IF bAlarmInit THEN
    bAlarmInit := FALSE; 
	fbSourceInfo.Clear();
	fbSourceInfo.sName:=wsLiteral_TO_UTF8(wsStationName);//'Machine';
	fbSourceInfo.nId:=iStationIndex;//83
	// Alarm_0610	610	Error	Siłownik przeciągania | Blokada wysunięcia - sprawdź czujnik lub odblokuj  
    arfbAlarm[0].CreateEx(stEventEntry := TC_EVENTS.AlarmClass.Alarm_0610, bWithConfirmation:= FALSE,  ipSourceInfo:= fbSourceInfo); 
	// Alarm_0611	611	Error	Siłownik przeciągania | Blokada wsunięcia - sprawdź czujnik lub odblokuj  
	arfbAlarm[1].CreateEx(stEventEntry := TC_EVENTS.AlarmClass.Alarm_0611, bWithConfirmation:= FALSE,  ipSourceInfo:= fbSourceInfo);
	// Alarm_0612	612	Error	Banda końcowa | Blokada wysunięcia - sprawdź czujnik lub odblokuj  
	arfbAlarm[2].CreateEx(stEventEntry := TC_EVENTS.AlarmClass.Alarm_0612, bWithConfirmation:= FALSE,  ipSourceInfo:= fbSourceInfo);
	// Alarm_0613	613	Error	Szlaban | Blokada wysunięcia - sprawdź czujnik lub odblokuj  
	arfbAlarm[3].CreateEx(stEventEntry := TC_EVENTS.AlarmClass.Alarm_0613, bWithConfirmation:= FALSE,  ipSourceInfo:= fbSourceInfo);
	// Alarm_0614	614	Error	Bład czujników przed przeciąganiem - sprawdź ułożenie formatek
	arfbAlarm[4].CreateEx(stEventEntry := TC_EVENTS.AlarmClass.Alarm_0614, bWithConfirmation:= FALSE,  ipSourceInfo:= fbSourceInfo);
	// Alarm_0615	615	Error	Bład czujników za przeciąganiem - sprawdź ułożenie formatek
	arfbAlarm[5].CreateEx(stEventEntry := TC_EVENTS.AlarmClass.Alarm_0615, bWithConfirmation:= FALSE,  ipSourceInfo:= fbSourceInfo);
	
END_IF

//CZYTANIE STATUSÓW
bStateError										:= (eState=E_Station.eError) OR (eState=E_Station.eResetting) OR NOT bEstop OR bIgnoreError;
tonEstopDelay									(IN:=bEStop,	PT:=T#4S);

IF bEnable AND tonEstopDelay.Q THEN
	// Alarm_0610	610	Error	Siłownik przeciągania | Blokada wysunięcia - sprawdź czujnik lub odblokuj  
	tonbDragOnSensor	(IN:= bDragActuator AND NOT bDragOnSensor	, PT:=T#2S);
	IF tonbDragOnSensor.Q THEN
		bHomingDone									:= FALSE;	
		//arfbAlarm[0].ipArguments.Clear() .AddString(stDrag.stError.sNcError);
		IF NOT arfbAlarm[0].bActive THEN
			arfbAlarm[0].Raise(nTimeStamp:=0);
		END_IF
	ELSE	
		IF  arfbAlarm[0].bActive AND bReset THEN
			arfbAlarm[0].Clear(nTimeStamp:=0, bResetConfirmation:= FALSE);
		END_IF	
	END_IF
	// Alarm_0611	611	Error	Siłownik przeciągania | Blokada wsunięcia - sprawdź czujnik lub odblokuj  
	tonbDragOffSensor	(IN:= NOT bDragActuator AND NOT bDragOffSensor	, PT:=T#2S);
	IF tonbDragOffSensor.Q THEN
		IF NOT arfbAlarm[1].bActive THEN
			arfbAlarm[1].Raise(nTimeStamp:=0);
		END_IF
	ELSE	
		IF  arfbAlarm[1].bActive AND bReset THEN
			arfbAlarm[1].Clear(nTimeStamp:=0, bResetConfirmation:= FALSE);
		END_IF	
	END_IF	
	// Alarm_0612	612	Error	Banda końcowa | Blokada wysunięcia - sprawdź czujnik lub odblokuj  
	tonbStoperOnSensor	(IN:= bStoperActuator AND NOT bStoperOnSensor	, PT:=T#2S);
	IF tonbStoperOnSensor.Q THEN
		IF NOT arfbAlarm[2].bActive THEN
			arfbAlarm[2].Raise(nTimeStamp:=0);
		END_IF
	ELSE	
		IF  arfbAlarm[2].bActive AND bReset THEN
			arfbAlarm[2].Clear(nTimeStamp:=0, bResetConfirmation:= FALSE);
		END_IF	
	END_IF	
	// Alarm_0613	613	Error	Szlaban | Blokada wysunięcia - sprawdź czujnik lub odblokuj  
	tonbGateSensor	(IN:= bGateActuator AND NOT bGateOnSensor	, PT:=T#2S);
	IF tonbGateSensor.Q THEN
		IF NOT arfbAlarm[3].bActive THEN
			arfbAlarm[3].Raise(nTimeStamp:=0);
		END_IF
	ELSE	
		IF  arfbAlarm[3].bActive AND bReset THEN
			arfbAlarm[3].Clear(nTimeStamp:=0, bResetConfirmation:= FALSE);
		END_IF	
	END_IF	
	// Alarm_0614	614	Error	Bład czujników przed przeciąganiem - sprawdź ułożenie formatek
	tonBeforeSensor	(IN:= NOT bFirstFormSensor AND bSecondFormSensor AND bConveyorBeforeRunning, PT:=T#20S);
	IF tonBeforeSensor.Q THEN
		IF NOT arfbAlarm[4].bActive THEN
			arfbAlarm[4].Raise(nTimeStamp:=0);
		END_IF
	ELSE	
		IF  arfbAlarm[4].bActive AND bReset THEN
			arfbAlarm[4].Clear(nTimeStamp:=0, bResetConfirmation:= FALSE);
		END_IF	
	END_IF	
	// Alarm_0615	615	Error	Bład czujników za przeciąganiem - sprawdź ułożenie formatek
	tonAfterSensor	(IN:= bAfterSensor AND bConveyorAfterRunning, PT:=T#20S);
	IF tonAfterSensor.Q THEN
		IF NOT arfbAlarm[5].bActive THEN
			arfbAlarm[5].Raise(nTimeStamp:=0);
		END_IF
	ELSE	
		IF  arfbAlarm[5].bActive AND bReset THEN
			arfbAlarm[5].Clear(nTimeStamp:=0, bResetConfirmation:= FALSE);
		END_IF	
	END_IF	
ELSE
	bError := FALSE;
END_IF

//******************PRZEJŚCIE DO eERROR*****************************

IF bError AND  NOT bStateError THEN
	eState 									:= E_Station.eError;
END_IF

//****************WYŚWIETLANIE STATUSU BLEDU************************
(*Wyświetlanie błedu na wyjściu*)
bError							:= FALSE;
FOR nAlarmNumerator := 0 TO 19 DO
	bError						:= bError OR arfbAlarm[nAlarmNumerator].bActive;
END_FOR

(*Przepisywanie nazwy stacji*)
sErrorStationName 							:= WSTRING_TO_STRING(wsStationName);
END_ACTION

ACTION Homing:


IF bHoming THEN // Bazowanie - podjazd do góry i ustawienie obrotu
	CASE iHomingCase OF
	
	0: 
		bHomingDone								:= FALSE;                                       		
		bDragActuator							:= FALSE;	
		bStoperActuator							:= TRUE; 	
		bGateActuator							:= FALSE;
			
		iHomingCase								:= 10;
	
	10: 
		iHomingCase								:= 20;
		
	20: 
		iHomingCase								:= 30;
		
		
	30:
		iHomingCase								:= 40;
		
	40:
		iHomingCase								:= 50;
	
	50: 
		iHomingCase								:= 60;
		
	60: 
		iHomingCase								:= 70;
	
	70:                             	
		iHomingCase								:= 80;

	80:
		iHomingCase								:= 100;

	100: //Zbazowano	
		iHomingCase								:= 0;
		eState									:= E_Station.eHomingDone;
	
	END_CASE
END_IF	
IF bHeightSet THEN

	bDragActuator								:= FALSE;	
	bStoperActuator								:= TRUE;
	bGateActuator								:= FALSE;
	eState										:= E_Station.eHomingDone;
		
END_IF
END_ACTION

ACTION Limits:
(*Wywowyłanie na początku*)


(*Prędkość zakręcania*)


(*Inny parametr*)
//...
END_ACTION

ACTION ManualMovements:

IF NOT bRun AND NOT bPrepare AND bManualMovement THEN
	bDragActuator							:=	bManualDragActuator;			
	bStoperActuator							:=	bManualStoperActuator;	
	bGateActuator							:=	bManualGateActuator;	
ELSE
	bManualDragActuator						:=	FALSE;		
	bManualStoperActuator					:=	TRUE;	
	bManualGateActuator						:=	FALSE;		
END_IF
	
IF bHoming OR bHeightSet THEN
	eState									:=	E_Station.eHoming;	
END_IF                                                	
                                                      	
Running();

IF NOT bRun AND NOT bPrepare THEN
	bCycleDone 								:= FALSE;
	bCycleNotDone 							:= FALSE;	
END_IF
END_ACTION

ACTION ResetAll:
(*****Reset bloczka*****)
IF bEnable THEN
	IF eState <> E_Station.eDisabled AND eState <> E_Station.ePreparingToDisable THEN
		IF bResetCycle THEN
			bResetCycleOn						:= TRUE;
			eState								:= E_Station.ePreparingToReady;
		END_IF
	END_IF
END_IF


IF bResetCycleOn THEN
	
	ResetCommands();
	eRunningState							:= E_DragStationState.eReady;	
	eState 				 					:= E_Station.eReady;

END_IF
END_ACTION

ACTION ResetCommands:
//KAsowanie komend ruchu 
                                                          	
bManualDragActuator								:=	FALSE;		
bManualStoperActuator							:=	FALSE;	
bManualGateActuator								:=	FALSE;	
                                                        	
bDragActuator									:=	FALSE;	
bStoperActuator									:=	TRUE;	
bGateActuator									:=	FALSE;
                                                          	
bResetCycleOn									:=	FALSE;	

iHomingCase										:=	0;
//bCycleDone								   	:=	FALSE;
END_ACTION

ACTION Running:
	
CASE eRunningState OF
	
	E_DragStationState.eDisabled:
		eRunningState								:= E_DragStationState.eReady; 
	
	E_DragStationState.eReady:

			//bDragActuator						:=	FALSE;
			//bStoperActuator					:=	TRUE;
			//bGateActuator						:=	FALSE;
			IF (bRun OR bPrepare) AND NOT bCycleDone THEN   
				eRunningState					:=	E_DragStationState.ePreparingToMove; 
       		END_IF

// Sygnal przygotowania do przeciaganiecia formatek		
	E_DragStationState.ePreparingToMove:
		bGateActuator							:=	TRUE;
		IF bGateOnSensor THEN
			eRunningState						:=	E_DragStationState.eLifting;
		END_IF
		
// Podnoszenie widel do przeciągania i sprawdzenie czy trafiły w otwór		
	E_DragStationState.eLifting:
	
		bStoperActuator							:=	FALSE;		
		IF NOT bStoperOnSensor AND bRun AND tonRunningLifting.Q THEN
			eRunningState						:=	E_DragStationState.eDraging;	
		END_IF
//  
	E_DragStationState.ePrepareToDrag:
		;
	
// Przeciąganie formatek
	E_DragStationState.eDraging:
	
		bDragActuator						:=	TRUE;
		IF bDragOnSensor THEN //100MS
			eRunningState							:= E_DragStationState.eDragingDone;
		END_IF

	E_DragStationState.eDragingDone:

		eRunningState							:= E_DragStationState.eEndingOfDrag;
	
	E_DragStationState.eEndingOfDrag:
		bDragActuator								:=	FALSE;
		IF bDragOffSensor THEN
			bStoperActuator							:=	TRUE;
			bGateActuator							:=	FALSE;				
			eRunningState							:= E_DragStationState.eEndingOfDragDone;
		END_IF	
		
	E_DragStationState.eEndingOfDragDone:
		
		eRunningState								:= E_DragStationState.eLowering;
	
	E_DragStationState.eLowering:
	
		eRunningState							:= E_DragStationState.eDraged;
	
	E_DragStationState.eDraged:
			
		eRunningState							:= E_DragStationState.eDragedDone;
		
	E_DragStationState.eDragedDone:
	
		bCycleDone									:= TRUE;	
		eRunningState								:= E_DragStationState.eReady;	
		
END_CASE
END_ACTION

ACTION Signals:

tonPreparingToReady		(IN:=	eState = E_Station.ePreparingToReady			,PT:= T#3S);
tonResetting			(IN:=	eState = E_Station.eResetting					,PT:= T#200MS);
tonHoming				(IN:=	eState = E_Station.eHoming						,PT:= T#1S);
rtResetCommands			(CLK:=	eState = E_Station.eReady 						,Q=>); 

tonRunningDraging		(IN:=	eRunningState = E_DragStationState.eDraging		,PT:= T#100MS);	//bylo 100
tonRunningLifting		(IN:=	eRunningState = E_DragStationState.eLifting		,PT:= T#100MS);	//bylo 100

tonRunningeEndingOfDrag	(IN:=	eRunningState = E_DragStationState.eEndingOfDrag 
								,PT:= T#5MS);								//100ms t#200ms

//Opóżnienie wysuwania przeciągania
tonNotDragActuatorDelay	(IN:=	NOT bDragActuator					,PT:=T#150MS);
END_ACTION

ACTION Statistics:
rtrigCycleTimerRead(CLK:=bCycleDone);
IF rtrigCycleTimerRead.Q THEN
	tCycleTime:=tonCycleTimer.ET;
END_IF
tonCycleTimer(IN:= eRunningState>E_DragStationState.eReady, PT:=T#1D);
END_ACTION

END_FUNCTION_BLOCK

// ---- POUs/P17_TurnTables.TcPOU
(*
Nazwa:			P14_TurnTable
Opis:			Stacja stołu obrotowego
Wersja:			v0.2
Data:			2024-11-06
Autor:			DP
Urzadzenia:		
Konfiguracja:	
Info:
- 4 wersja z safety po EC

*)
PROGRAM P17_TurnTables
VAR_INPUT
	IbExitTurnTableAfterSensor 			:BOOL;
	IbExitTurnTablePackageSensor 	AT %I*	:BOOL;		
END_VAR
VAR
	
	(*********STOL ODBIERAJACY*******************)
	
	tonIbExitTurnTable1Working		: TON;
	fbTurnTable						: FB_MitsubishiInverter; 	//Bloczek do obsługi falownika stołu obrotewego
	eTurnTableState					: E_Station;
	eTurnTableRunningState			: E_ConveyorState;
	fbTurnTableState				: FB_State;

	uiTurnTableSW					AT %I*: UINT;
	uiTurnTableActualVelocity		AT %I*: UDINT;
	uiTurnTableCW  					AT %Q*: UINT;
	udiTurnTableVelocity			AT %Q*: UDINT;	
	
	tonIbTurnTableCycleStopButton	: TON;
	bExitTurnTableCmdStartDelay		: BOOL;
	tonbExitTurnTableCmdStartDelay	: TON;
	
	//fbExitConveyor					: FB_LenzeInverter;
	fbExitConveyor					: FB_MitsubishiInverter;
	QnExitConveyorVelocitySV 		AT %Q*: UDINT; 		
	InExitConveyorVelocityCV 		AT %I*: UDINT;	
	InExitConveyorSTW 				AT %I*: UINT; 
	QnExitConveyorConvCTW 			AT %Q*: UINT;  			
	InExitConveyorErrorCode 		AT %I*:UINT;			

	fbExitTurnTableGate				: FB_Gate;				// Bloczek obsługi gata	
	QbExitTurnTableGate 			: BOOL; 				// Wyjście sterujące szlabanem stołu odbiorczego
	
	
	tonbExitTurnTableCmdStart		: TON;
	tonIbExitTurnTableAfterSensor	: TON;
	tonbExitTurnTableGateRunOn		: TON;
	tonbExitTurnTableGateRunOff		: TON;	
	
	fbExitConveyorGate				: FB_Gate;				
	QbExitConveyorGate 				AT %Q*: BOOL;			
	IbExitConveyorGateAfterSensor 	AT %I*: BOOL;		//Blizej szlabanu
	IbExitConveyorGateAfterSensor2 	AT %I*: BOOL;		//Dalej szlabanu
	
	
END_VAR

aTurnTable();
aConveyor();
aConveyorGate();
aTurnTableGate();
aTurnTableGateLogic();
(*
tonIbTurnTableCycleStopButton	(IN:=NOT IbTurnTableCycleStopButton AND bExitTurnTableCmdStart AND NOT (P00_PackML.fbPMLAuto.ePMLState = Tc3_PackML.E_PMLState.ePMLState_EXECUTE), PT:=T#10MS);
IF tonIbTurnTableCycleStopButton.Q THEN
	bExitTurnTableCmdStartDelay	:=	TRUE;
END_IF
IF bExitTurnTableCmdStartDelay THEN
	bExitTurnTableCmdStart	:=	FALSE;
END_IF
tonbExitTurnTableCmdStartDelay		(IN:= bExitTurnTableCmdStartDelay, PT:=T#5S);
IF 	tonbExitTurnTableCmdStartDelay.Q THEN
	bExitTurnTableCmdStartDelay	:=	FALSE;
END_IF
*)

IbTurnTableMotorOK							;
IbTurnTableEmergencyStopButtonPressed	;
IbTurnTableCycleStartButton				;
IbTurnTableCycleStopButton				;
										;

P00_Signalization.QbTurnTableStartLamp;							
P00_Signalization.QbTurnTableResetLamp;

ACTION aConveyor:
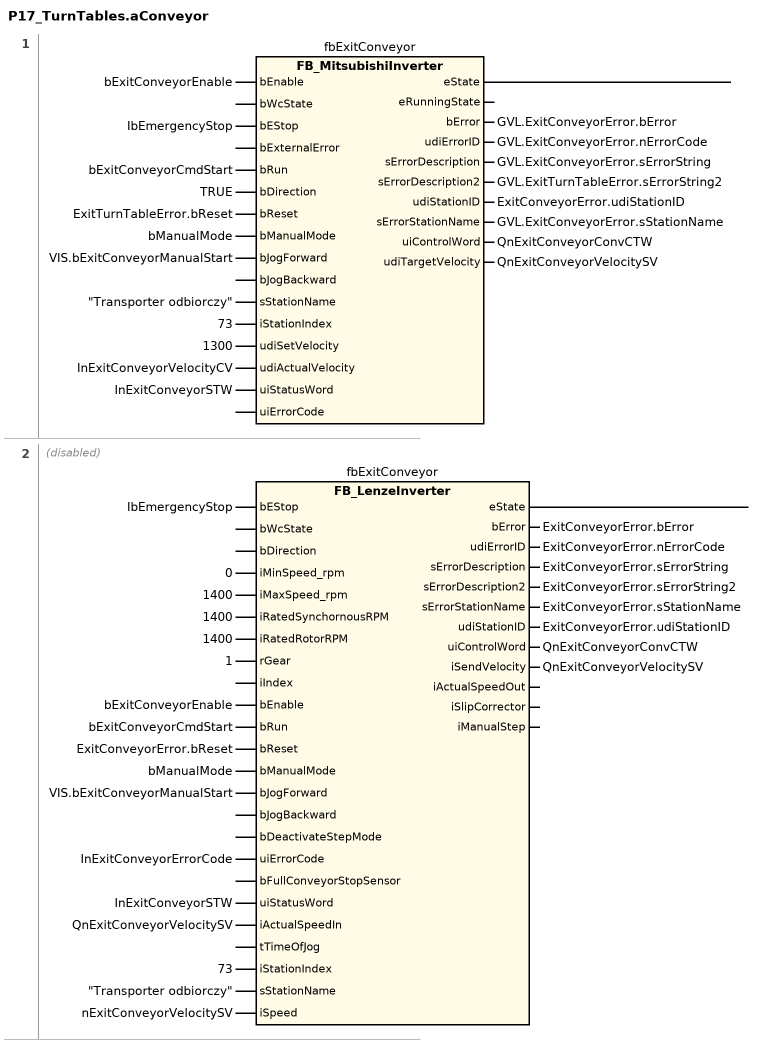
// NETWORK 1
fbExitConveyor(
    bEnable := bExitConveyorEnable,
    bEStop := IbEmergencyStop,
    bRun := bExitConveyorCmdStart,
    bDirection := TRUE,
    bReset := ExitTurnTableError.bReset,
    bManualMode := bManualMode,
    bJogForward := VIS.bExitConveyorManualStart,
    sStationName := "Transporter odbiorczy",
    iStationIndex := 73,
    udiSetVelocity := 1300,
    udiActualVelocity := InExitConveyorVelocityCV,
    uiStatusWord := InExitConveyorSTW,
    bError => GVL.ExitConveyorError.bError,
    udiErrorID => GVL.ExitConveyorError.nErrorCode,
    sErrorDescription => GVL.ExitConveyorError.sErrorString,
    sErrorDescription2 => GVL.ExitTurnTableError.sErrorString2,
    udiStationID => ExitConveyorError.udiStationID,
    sErrorStationName => GVL.ExitConveyorError.sStationName,
    uiControlWord => QnExitConveyorConvCTW,
    udiTargetVelocity => QnExitConveyorVelocitySV); // FB_MitsubishiInverter

// NETWORK 2 (disabled)
// fbExitConveyor(
//     bEStop := IbEmergencyStop,
//     iMinSpeed_rpm := 0,
//     iMaxSpeed_rpm := 1400,
//     iRatedSynchornousRPM := 1400,
//     iRatedRotorRPM := 1400,
//     rGear := 1,
//     bEnable := bExitConveyorEnable,
//     bRun := bExitConveyorCmdStart,
//     bReset := ExitConveyorError.bReset,
//     bManualMode := bManualMode,
//     bJogForward := VIS.bExitConveyorManualStart,
//     uiErrorCode := InExitConveyorErrorCode,
//     uiStatusWord := InExitConveyorSTW,
//     iActualSpeedIn := QnExitConveyorVelocitySV,
//     iStationIndex := 73,
//     sStationName := "Transporter odbiorczy",
//     iSpeed := nExitConveyorVelocitySV,
//     bError => ExitConveyorError.bError,
//     udiErrorID => ExitConveyorError.nErrorCode,
//     sErrorDescription => ExitConveyorError.sErrorString,
//     sErrorDescription2 => ExitConveyorError.sErrorString2,
//     sErrorStationName => ExitConveyorError.sStationName,
//     udiStationID => ExitConveyorError.udiStationID,
//     uiControlWord => QnExitConveyorConvCTW,
//     iSendVelocity => QnExitConveyorVelocitySV); // FB_LenzeInverter
END_ACTION

ACTION aConveyorGate:
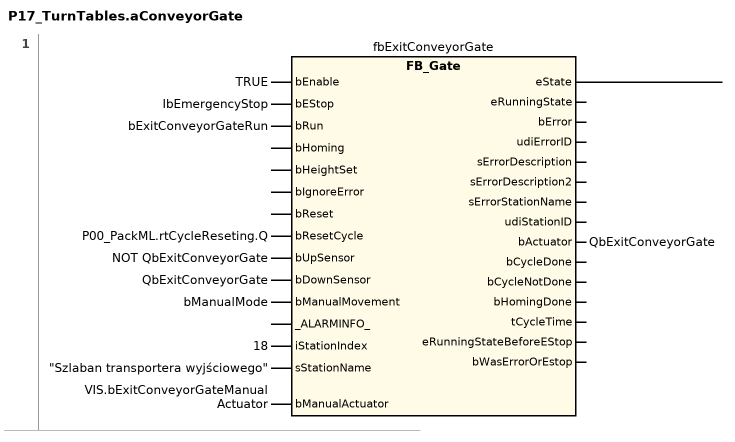
// NETWORK 1
fbExitConveyorGate(
    bEnable := TRUE,
    bEStop := IbEmergencyStop,
    bRun := bExitConveyorGateRun,
    bResetCycle := P00_PackML.rtCycleReseting.Q,
    bUpSensor := NOT QbExitConveyorGate,
    bDownSensor := QbExitConveyorGate,
    bManualMovement := bManualMode,
    iStationIndex := 18,
    sStationName := "Szlaban transportera wyjściowego",
    bManualActuator := VIS.bExitConveyorGateManualActuator,
    bActuator => QbExitConveyorGate); // FB_Gate
END_ACTION

ACTION aTurntable:
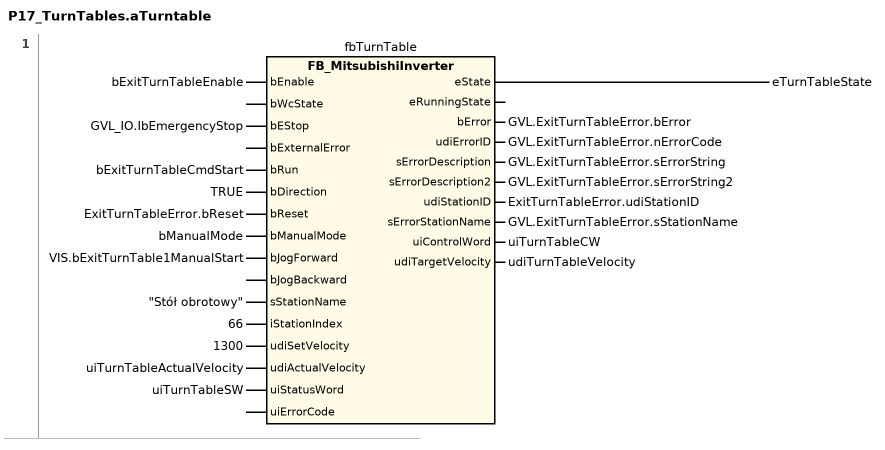
// NETWORK 1
fbTurnTable(
    bEnable := bExitTurnTableEnable,
    bEStop := GVL_IO.IbEmergencyStop,
    bRun := bExitTurnTableCmdStart,
    bDirection := TRUE,
    bReset := ExitTurnTableError.bReset,
    bManualMode := bManualMode,
    bJogForward := VIS.bExitTurnTable1ManualStart,
    sStationName := "Stół obrotowy",
    iStationIndex := 66,
    udiSetVelocity := 1300,
    udiActualVelocity := uiTurnTableActualVelocity,
    uiStatusWord := uiTurnTableSW,
    bError => GVL.ExitTurnTableError.bError,
    udiErrorID => GVL.ExitTurnTableError.nErrorCode,
    sErrorDescription => GVL.ExitTurnTableError.sErrorString,
    sErrorDescription2 => GVL.ExitTurnTableError.sErrorString2,
    udiStationID => ExitTurnTableError.udiStationID,
    sErrorStationName => GVL.ExitTurnTableError.sStationName,
    uiControlWord => uiTurnTableCW,
    udiTargetVelocity => udiTurnTableVelocity); // FB_MitsubishiInverter
eTurnTableState := fbTurnTable.eState;
END_ACTION

ACTION aTurntableGate:
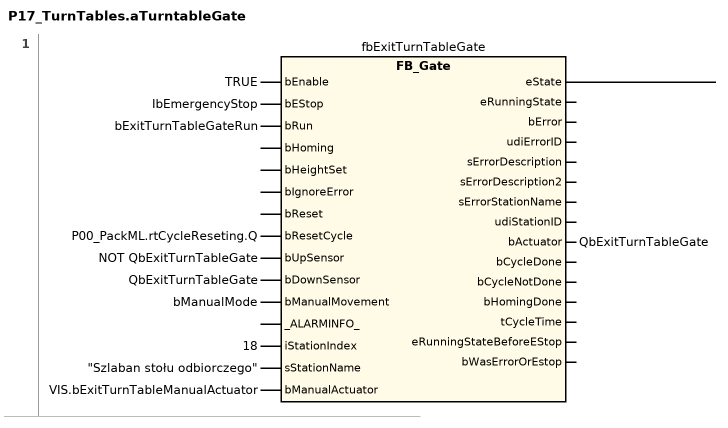
// NETWORK 1
fbExitTurnTableGate(
    bEnable := TRUE,
    bEStop := IbEmergencyStop,
    bRun := bExitTurnTableGateRun,
    bResetCycle := P00_PackML.rtCycleReseting.Q,
    bUpSensor := NOT QbExitTurnTableGate,
    bDownSensor := QbExitTurnTableGate,
    bManualMovement := bManualMode,
    iStationIndex := 18,
    sStationName := "Szlaban stołu odbiorczego",
    bManualActuator := VIS.bExitTurnTableManualActuator,
    bActuator => QbExitTurnTableGate); // FB_Gate
END_ACTION

ACTION aTurnTableGateLogic:
//Jeżeli stół pracuje 
bExitTurnTableCmdStart;
//To ruszaj szlabanem
bExitTurnTableGateRun;
//Czujnik na szlabanie etykieciarki:
IbExitTurnTableAfterSensor;

tonbExitTurnTableCmdStart		(IN:=bExitTurnTableCmdStart,											PT:=T#3S);
tonIbExitTurnTableAfterSensor	(IN:=IbExitTurnTableAfterSensor,										PT:=T#3S);
tonbExitTurnTableGateRunOn		(IN:=bExitTurnTableGateRun ,											PT:=T#5S);
tonbExitTurnTableGateRunOff		(IN:=NOT bExitTurnTableGateRun AND tonIbExitTurnTableAfterSensor.Q,		PT:=T#5S);//bylo 1

IF tonbExitTurnTableCmdStart.Q THEN
	bExitTurnTableGateRun R= tonbExitTurnTableGateRunOn.Q;
	bExitTurnTableGateRun S= tonbExitTurnTableGateRunOff.Q;	
END_IF
END_ACTION

END_PROGRAM

// ---- POUs/FB/FB_LenzeInverter.TcPOU
////////////////////////////////////////////////////////////////////////////////////////////////////////////
(*	TKMatik
	Blok funkcyjny, sterujacy falownikiem firmy Lenze model:i550
	v.1.3 16.01.2019
	v.1.4 22.08.2019
	v.1.5 29.07.2020
	Wymagane pliki: E_Station (ENUM)
	Data modyfikacji: 29.07.2020
	
	--->Obsluga bloku:
	Blok umozliwia sterownie falownikiem Lenze i550 w trybie manulanym i automatycznym
	*TRYB AUTOMATYCZNY*
	Po podaniu sygnalu wysokiego na wejscie bEnable rozoczyna sie procedura uruchamiania falownika
	Wejscie bRun umozliwiaja odpowiednio uruchomienie silnika i jego zatrzymanie 
	Wejscie bReset umozliwa wykonanie procedury resetu bloku i bledu falownika
	Wejscia iMinSpeed_rpm oraz iMaxSpeed_rpm pozwalaja na programowe ograniczenie obrotow silnika
	Wejscie iSpeed sluzy zadawania wartosci predkosci
	Mozliwa jest rowniez zmiana kierunku obrotow silnika przy pomocy wejscia bDirection
	*TRYB MANULANY*
	Sterowanie w trybie manulanym opiera sie o wykrywanie czasu przyciniecia przyciku
	Dla krotkiego przycisniecia wykonywany jest ruch silnika o krok ktorego czas musi byc zadany na wejscie bloku - opcje ta mozna dezaktywowac wejsciem bStepModeNotActive
	Dla dlugiego przycisniecia ruch jest wykonywany do czasu zaprzestania naciskania przycisku
	
	
	Wejscia bloku, ktore nalezy polinkowac ze zmiennymi falownika:
		-uiErrorCode
		-uiStatusWord
		-ActualSpeed 
	Wyjscia bloku, ktore nalezy polinkowac ze zmiennymi falownika:
		-uiControlWord
		-iSendVelocity
*)
////////////////////////////////////////////////////////////////////////////////////////////////////////////

FUNCTION_BLOCK FB_LenzeInverter

VAR_INPUT
	bEStop														: BOOL;													// Pozwolenie na prace bloku z SAFETY (TRUE-maszyna gotowa do pracy FALSE-brak pozolenia na prace)
	bWcState													: BOOL;													// Zmienna WcState - TRUE w przypadku odebrania niewlasciwej ramki EtherCAT
	bDirection													: BOOL;													// Kierunek obrotow silnika 
	iMinSpeed_rpm												: INT				:= 1000;							// Minimalna prędkość obrotowa
	iMaxSpeed_rpm												: INT				:= 2840;							// Maksymalna prędkość obrotowa
	iRatedSynchornousRPM										: INT				:= 3000;							// Predkosc synchorniczna (wzor: RatedSynchronousRPM = 60 * Frequency / NumberOfPolePair)
	iRatedRotorRPM												: INT				:= 2840;							// Znamionowe obroty silnika
	rGear														: REAL;													// Przekładnia
	iIndex														: INT;													// Indeks falownika
	bEnable														: BOOL;													// Uruchomienie bloku
	bRun														: BOOL;													// Komenda na uruchomienie 
	bReset														: BOOL;													// Reset falownika po bledzie
	bManualMode													: BOOL;													// Tryb manualny
	bJogForward													: BOOL;													// Komenda na ruch w kierunku dodatnim 
	bJogBackward												: BOOL;													// Komenda na ruch w kierunku ujemnym 
	bDeactivateStepMode											: BOOL;													// Zmienna dezaktywujaca przesuwanie silnika o krok po nacisnieciu JOGa
	uiErrorCode 				(*Devices*)						: UINT;													// Kod bledu falownika
	bFullConveyorStopSensor										: BOOL;													// Zatrzymanie transportera ze względu zapełnienia
	uiStatusWord				(*Devices*)						: UINT;													// Status wysylany z falownika
	iActualSpeedIn				(*Devices*)						: INT;													// Zmienna z falownika przepisana na wyjscie do zmiennej QiActualSpeed
	tTimeOfJog													: TIME				:= T#2S;
	iStationIndex												: UDINT;												// Numer stacji 
	sStationName												: WSTRING;												// Nazwa stacji
	iSpeed														: INT;													// Predkosc zadana przypisana do zmiennej Qn_SV wysylanej do falownika  
END_VAR                                                                         			                    		
VAR_OUTPUT                                                                      			                    		
	eState														: E_Station;											// Stan pracy bloku
	
	bError														: BOOL;													// Blad falownika
	udiErrorID													: UDINT;												// Nr błędu bloku funkcyjnego
	sErrorDescription											: STRING(200);											// Opis błędu
	sErrorDescription2											: STRING(200);											// Opis błędu
	sErrorStationName											: STRING;												// Nazwa stacji
	udiStationID												: UDINT;				// Nr stacji	
	uiControlWord(*Wymaga przypisania do urządzenia*)			: UINT;													// ControlWord wysylany do falownika 
	iSendVelocity(*Wymaga przypisania do urządzenia*)			: INT;													// Wartosc predkosci zadanej wysylanej do falownika
	iActualSpeedOut												: INT;													// Wartosc predkosci akutalnej przepisanej z wyjscia
	iSlipCorrector												: INT;													// Wspolczynnik korygujacy wartosc poslizgu
	iManualStep													: INT;
END_VAR                                     					
VAR                                         					
	rtRun														: R_TRIG;												// Triger rozpoczynajacy obrot osi silnika
	ftReset														: F_TRIG;												// Triger zbocza opadajacego resetu
	rtInvertDirection											: R_TRIG;												// Triger zmieniajacy kierunek obrotu osi silnika
	ftInvertDirection											: F_TRIG; 												// Triger zbocza opadajacego od zmiany kierunku                                      		                                                                                                          		                 											                                		
	rtJogForward												: R_TRIG;												// Trigger wykrywajacy zbocze narasatace komendy ruchu w kierunku dodatnim w trybie manulanym
	rtJogBackward												: R_TRIG;												// Trigger wykrywajacy zbocze narasatace komendy ruchu w kierunku ujemnym w trybie manulanym
	ftJogForward												: F_TRIG;												// Trigger wykrywajacy zbocze opadajace komendy ruchu w kierunku dodatnim w trybie manulanym
	ftJogBackward												: F_TRIG;												// Trigger wykrywajacy zbocze opadajace komendy ruchu w kierunku ujemnym w trybie manulanym
                                     					
	tonTimeOfJog												: TON;													// Timer odliczajacy czas trwania ruchu silnika w trybie manualnym
	tonPressing													: TON;													// Timer odliczajacy czas nacisniecia przycisku w trybie manulanym
	
    iCalculateVelocity											: INT;													// Wartosc predkosci wykorzystwanej do obliczen w bloku                                  	                                                                		
	
	bCheckInitTimeError											: BOOL;													// Blad oczekiwania na odpowiedz falownika
	tonCheckInitTime											: TON;													// Timer odliczajacy czas odpowiedzi falownika
	
	bWcStateError												: BOOL;													// Blad zmiennej WcState - odczytanie blednej ramki danych przez urzadzenie EtherCAT
	
	bLenzeReadiness												: BOOL;													// Gotowosc falownika do pracy na podstawie bitu StatusWord --> SwitchedOn
	bLenzeReadinessError										: BOOL;													// Blad zwiazany z utraceniem gotowosci do pracy przez falownik
	bFullConveyorError											: BOOL;														// Blad zwiazany z przepełnieniem transportera
	
	
	iPreparingStep												: INT;													// Krok procedury przygotowania do pracy falownika
	
	
	(*Zmienne ControlWord*)
	bSwitchOn													: BOOL;													// Zalacz falownik do trybu gotowsci
	bEnableVoltage												: BOOL;													// Zalacz zasilanie na zaciski falownika
	bQuickStop													: BOOL;													// Bezpieczne zatrzymanie
	bEnableOperation											: BOOL;													// Rozpoczecie pracy falownika
	bOperationModeSpecific1										: BOOL;
	bOperationModeSpecific2										: BOOL;
	bOperationModeSpecific3										: BOOL;
	bFaultReset													: BOOL;													// Reset bledu
	bHalt														: BOOL;													// Zatrzymanie procesowe
	bOperationModeSpecific4										: BOOL;
	bReserved1													: BOOL;
	bReserved2													: BOOL;
	bReserved3													: BOOL;
	bReserved4													: BOOL;
	bHoldingBrakeRelease										: BOOL;
	bReserved5													: BOOL;
	                                        					
	(*Zmienne StatusWord*)                  					
	bReadyToSwitchOn											: BOOL;													// Gotowy na zalaczenie do trybu gotowosci
	bSwitchedOn													: BOOL;													// Zalaczony w tryb gotowosci do pracy
	bOperationEnabled											: BOOL;													// Wykonywanie pracy
	bFaultActive												: BOOL;													// Akytwny blad falownika
	bVoltageEnabled												: BOOL;													// Zalaczone zasilanie na zaciski falownika
	bQuickStopActive											: BOOL;													// Aktywne bezpieczne zatrzymanie				
	bSwitchOnDisabled											: BOOL;													// Tryb nieaktywnosci falownika	
	bWarningActive												: BOOL;													// Aktywne ostrzezenie falownika
	bDeactiveRPDOs												: BOOL;
	bRemote														: BOOL;													// Mozliwosc wykonyania operacji
	bTargetReached												: BOOL;													// Osiagniecie predkosci zadanej
	bInternalLimitActive										: BOOL;
	bReserved6													: BOOL;
	bReserved7													: BOOL;
	bBreakeReleased												: BOOL;
	bSTONotActive												: BOOL;													// Bezpieczne zatrzymanie nieaktywne
	
	rLenzeGear													: REAL;
	
			//Zmienne od EVENTLOGGER
	bAlarmInit 						: BOOL := TRUE; 
	nAlarmNumerator					: INT;
	arfbAlarm						: ARRAY[0..19] OF  FB_TcAlarm;		//Tablica bloczków błędów
	fbSourceInfo 					: FB_TcSourceInfo;
	iSourceInfo						: I_TcSourceInfo;
	sAlarmTest						: STRING;
	//Koniec zmiennych od EVENTLOGGER
END_VAR

VAR_IN_OUT
 
END_VAR


(*Status WORD:													
	Bit 0: Ready to switch on
	Bit 1: Switched on
	Bit 2: Operation enabled
	Bit 3: Fault active
	Bit 4: Voltage enabled
	Bit 5: Quick stop
	Bit 6: Switch on disabled
	Bit 7: Warning active
	Bit 8: Deactivate RPDOs
	Bit 9: Remote
	Bit 10: Target speed reached
	Bit 11: Internal limit active
	Bit 12: Reserved
	Bit 13: Reserved
	Bit 14: Brake released
	Bit 15: Safe torque off (STO) not active*)
				
	(*Control WORD:
	Bit 0: Switch On
	Bit 1: Enable Voltage
	Bit 2: Activate quick Stop
	Bit 3: Enable operation
	Bit 4: Operation mode specific
	Bit 5: Operation mode specific
	Bit 6: Operation mode specific
	Bit 7: Fault reset
	Bit 8: Halt
	Bit 9: Operation mode specific
	Bit 10: Reserved
	Bit 11: Reserved
	Bit 12: Reserved
	Bit 13: Reserved
	Bit 14: Holding brake release
	Bit 15: Reserved*)

ACT_EStop();
ACT_StatusWord();																										// Przypisanie bitow StatusWorda do zmiennych
ACT_ErrorHandling();
aStationID();

rtRun															(CLK:= bRun);
rtJogForward													(CLK:= bJogForward);
rtJogBackward													(CLK:= bJogBackward);
ftJogForward													(CLK:= bJogForward);
ftJogBackward													(CLK:= bJogBackward);
                                                               
                                                                
IF 	NOT bEnable 												AND 
	bEStop 														AND  
	eState <> E_Station.eAborting 								AND 
	eState <> E_Station.eAborting 								THEN
	
	eState:= E_Station.ePreparingToDisable;
END_IF


		
CASE eState OF
	
	E_Station.ePreparingToDisable: (*Przygotowanie do wylaczenia*)
	
		bQuickStop 												:= FALSE;
		bEnableVoltage											:= FALSE;
		bSwitchOn												:= FALSE;
		bEnableOperation 										:= FALSE;
		bFaultReset												:= FALSE;
		tonTimeOfJog.IN											:= FALSE;
		tonPressing.IN											:= FALSE;
		iPreparingStep											:= 0;
		iManualStep												:= 0;
		
		bLenzeReadinessError									:= FALSE;
		bFullConveyorError										:= FALSE;
		bWcStateError											:= FALSE;
		bCheckInitTimeError										:= FALSE;
		                                         
		eState:= E_Station.eDisabled;

		
	E_Station.eDisabled: (*Stan nieaktywnosci falowika*)
	
		IF bEnable THEN																									// Rozpoczecie proceduru uruchomienia falownika 								
			eState:= E_Station.ePreparingToReady;	                                		                                							
		END_IF                                      		                                							
	
			                                    		                                													
	E_Station.ePreparingToReady: (*Przygotwanie do gotowosci*)
	
	
		CASE iPreparingStep OF
			0:
				bSwitchOn										:= FALSE;
			    bEnableVoltage	                                := FALSE;
			    bQuickStop		                                := FALSE;
			    bEnableOperation                                := FALSE;
				iPreparingStep:= 10;
				
				IF bSwitchedOn THEN
					iPreparingStep:= 30;
				END_IF
				
			10:
				IF bSwitchOnDisabled THEN
					bEnableVoltage								:= TRUE;
					bQuickStop									:= TRUE;
					iPreparingStep:= 20;
				END_IF
			
			20:
				IF bReadyToSwitchOn THEN
					bSwitchOn									:= TRUE;
					iPreparingStep:= 30;
				END_IF
			
			30:
				IF bSwitchedOn THEN
					iPreparingStep:= 0;
					eState:= E_Station.eReady;
				END_IF
				
				
		END_CASE
	
			
	E_Station.eReady:	(*Gotowosc i oczekiwanie na komendy*)

		IF rtRun.Q THEN
			bEnableOperation									:= TRUE;
			eState:= E_Station.eStarting;
		END_IF
		
		IF bManualMode THEN
			iManualStep:= 0;
			eState:= E_Station.eManualMovement;
		END_IF
														
		
		
	E_Station.eStarting: (*Stan rozpoczynania pracy falownika*)
	
		IF bOperationEnabled THEN
			eState:= E_Station.eRunning;
		END_IF
		
		IF NOT bRun THEN
			bEnableOperation									:= FALSE;									
			eState:= E_Station.eStopping;
		END_IF
		
				
	E_Station.eRunning: (*Stan wykonywania pracy falownika*)
	
		IF NOT bRun THEN
			bEnableOperation									:= FALSE;									
			eState:= E_Station.eStopping;
		END_IF
		
			
	E_Station.eStopping:
	
		IF NOT bOperationEnabled THEN
			eState:= E_Station.eReady;
		END_IF
		
				
	E_Station.eAborting: (*Stan bezpiecznego zatrzymywania silnika*)	
	
		bQuickStop 												:= FALSE;
	    bEnableVoltage											:= FALSE;
	    bSwitchOn												:= FALSE;
		bEnableOperation 										:= FALSE;
		
		tonTimeOfJog.IN											:= FALSE;
		tonPressing.IN											:= FALSE;
		iManualStep												:= 0;
		iPreparingStep											:= 0;
		
		
		eState:= E_Station.eAborted;
		
		
	E_Station.eAborted: (*Stan bezpiecznego zatrzymania silnika*)
	                              			
		IF bEstop THEN
			IF NOT bError THEN
				IF bEnable THEN
					eState:= E_Station.ePreparingToReady;
				ELSE
					eState:= E_Station.ePreparingToDisable;
				END_IF
			ELSE 
				eState:= E_Station.eError;	
			END_IF	
		END_IF
		
					
	E_Station.eError: (*Stan bledu*)
													
		bQuickStop 												:= FALSE;
		bEnableVoltage											:= FALSE;
		bSwitchOn												:= FALSE;
		bEnableOperation 										:= FALSE;
		
		tonTimeOfJog.IN											:= FALSE;
		tonPressing.IN											:= FALSE;
		iManualStep												:= 0;
		iPreparingStep											:= 0;

		IF bReset THEN
			IF bCheckInitTimeError THEN
				bCheckInitTimeError								:= FALSE;
			END_IF
			IF bWcStateError THEN
				bWcStateError									:= FALSE;
			END_IF
			IF bLenzeReadinessError THEN
				bLenzeReadinessError							:= FALSE;
			END_IF
			IF 	bFullConveyorError	THEN
				bFullConveyorError								:= FALSE;
			END_IF
		END_IF
		
		bFaultReset												:= bReset; 

		
		IF NOT bError THEN 
			
			bFaultReset											:= FALSE;
		
			eState:= E_Station.ePreparingToReady;	
				
		END_IF
		
		
	E_Station.eManualMovement: (*Stan wykonywania ruchow manualnych*)
		
		ACT_ManualMovements();
		
									
END_CASE



IF ABS(iActualSpeedIn) > iSlipCorrector THEN
	IF iActualSpeedIn > 0 THEN
		iActualSpeedOut													:= (iActualSpeedIn - iSlipCorrector) / REAL_TO_INT(rGear);					// Przepisanie wartosci z wejscia bloku na jego wyjscie		
	ELSE
		iActualSpeedOut													:= (iActualSpeedIn + iSlipCorrector) / REAL_TO_INT(rGear);					// Przepisanie wartosci z wejscia bloku na jego wyjscie	
	END_IF
ELSE
	iActualSpeedOut													:= 0;
END_IF										


ACT_Calculations();	
ACT_ControlWord();																									//Przypisanie zmiennych do bitow ControlWorda


tonPressing();																								
tonTimeOfJog();

ACTION ACT_Calculations:
                                                    		
(*IF ABS(iSpeed) < iMinSpeed_rpm THEN																						// Warunki programowaego ograniczenia predkosci do wartosci min i max
	iSpeed 														:= iMinSpeed_rpm;
END_IF                                                  		
IF ABS(iSpeed) > iMaxSpeed_rpm THEN                     		
	iSpeed														:= iMaxSpeed_rpm;
END_IF                                                  	
*)//dp
                                                   	
IF bDirection THEN																										                                    	
	iCalculateVelocity											:= -iSpeed;
ELSE                                                    	
	iCalculateVelocity											:= iSpeed;
END_IF

(*Ruchy manualne JOG definuja kierunek ruchu niezaleznie od bDirection*)		
IF bJogForward THEN
	iCalculateVelocity											:= iSpeed;
ELSIF bJogBackward THEN
	iCalculateVelocity											:= -iSpeed;
END_IF
	

iSlipCorrector													:= iRatedSynchornousRPM - iRatedRotorRPM;				// Obliczenie wspolczynnika korygujacego wartosc poslizgu


(*Kontrola poprawności parametryzacji przekładni*)
IF rGear < 1 THEN
	rLenzeGear													:= 1;
ELSE
	rLenzeGear													:= rGear;
END_IF


(*Korekcja wartosci zadanej predkosci o wartosc poslizgu*)
IF iCalculateVelocity >= 0 THEN
	iSendVelocity												:= (iCalculateVelocity * REAL_TO_INT(rLenzeGear)) + iSlipCorrector ;
ELSIF iCalculateVelocity <0 THEN
	iSendVelocity												:= (iCalculateVelocity * REAL_TO_INT(rLenzeGear)) - iSlipCorrector;
END_IF
END_ACTION

ACTION ACT_ControlWord:
uiControlWord.0 								:= bSwitchOn;
uiControlWord.1 								:= bEnableVoltage;
uiControlWord.2 								:= bQuickStop;
uiControlWord.3 								:= bEnableOperation;
uiControlWord.4 								:= bOperationModeSpecific1;
uiControlWord.5 								:= bOperationModeSpecific2;
uiControlWord.6 								:= bOperationModeSpecific3;
uiControlWord.7 								:= bFaultReset;
uiControlWord.8 								:= bHalt;
uiControlWord.9 								:= bOperationModeSpecific4;
uiControlWord.10 								:= bReserved1;
uiControlWord.11 								:= bReserved2;
uiControlWord.12 								:= bReserved3;
uiControlWord.13 								:= bReserved4;
uiControlWord.14 								:= bHoldingBrakeRelease;
uiControlWord.15 								:= bReserved5;
END_ACTION

ACTION ACT_ErrorHandling:
// Alarm_0580	580	Error	Zresetuj błąd na panelu falownika {0}
// Alarm_0581	581	Error	Błąd komunikacji z urządzeniem (WcState)
// Alarm_0582	582	Error	Utracono gotowość falownika do pracy
// Alarm_0583	583	Error	Przekroczenie czasu oczekiwania na odpowiedź falownika
// Alarm_0584	584	Error	Przepełnienie

IF bAlarmInit THEN
    bAlarmInit := FALSE; 
	fbSourceInfo.Clear();
	fbSourceInfo.sName:=wsLiteral_TO_UTF8(sStationName);//'Machine';
	fbSourceInfo.nId:=iStationIndex;//2700;
	// Alarm_0580	580	Error	Zresetuj błąd na panelu falownika {0}
    arfbAlarm[0].CreateEx(stEventEntry := TC_EVENTS.AlarmClass.Alarm_0580, bWithConfirmation:= FALSE,  ipSourceInfo:= fbSourceInfo); 
	// Alarm_0581	581	Error	Błąd komunikacji z urządzeniem (WcState)
	arfbAlarm[1].CreateEx(stEventEntry := TC_EVENTS.AlarmClass.Alarm_0581, bWithConfirmation:= FALSE,  ipSourceInfo:= fbSourceInfo);
	// Alarm_0582	582	Error	Utracono gotowość falownika do pracy
	arfbAlarm[2].CreateEx(stEventEntry := TC_EVENTS.AlarmClass.Alarm_0582, bWithConfirmation:= FALSE,  ipSourceInfo:= fbSourceInfo);
	// Alarm_0583	583	Error	Przekroczenie czasu oczekiwania na odpowiedź falownika
	arfbAlarm[3].CreateEx(stEventEntry := TC_EVENTS.AlarmClass.Alarm_0583, bWithConfirmation:= FALSE,  ipSourceInfo:= fbSourceInfo);
	// Alarm_0584	584	Error	Przepełnienie
	arfbAlarm[4].CreateEx(stEventEntry := TC_EVENTS.AlarmClass.Alarm_0584, bWithConfirmation:= FALSE,  ipSourceInfo:= fbSourceInfo);
	
END_IF



tonCheckInitTime.IN												:= eState = E_Station.ePreparingToReady OR eState = E_Station.eStarting OR eState = E_Station.eStopping;																														
tonCheckInitTime.PT												:= T#5S;
tonCheckInitTime();                                     		

IF tonCheckInitTime.Q THEN
	bCheckInitTimeError											:= TRUE;
END_IF  

IF bWcState THEN
	bWcStateError												:= TRUE;
END_IF   

IF bFullConveyorStopSensor THEN
	bFullConveyorError:= TRUE;
END_IF

bLenzeReadiness													:= bSwitchedOn;

IF NOT bLenzeReadiness THEN
	IF 	eState = E_Station.eReady				OR
		eState = E_Station.eStarting			OR
		eState = E_Station.eRunning				OR
		eState = E_Station.eStopping			OR
		eState = E_Station.eManualMovement		THEN

		bLenzeReadinessError									:= TRUE;
		
	END_IF                                                		
END_IF    

                                         	                                                        	                                                     	
//bError															:= bFaultActive OR bCheckInitTimeError OR bWcStateError OR bLenzeReadinessError OR bFullConveyorError;

// Alarm_0580	580	Error	Zresetuj błąd na panelu falownika {0}
IF bFaultActive AND bEnable THEN
	arfbAlarm[0].ipArguments.Clear() .AddUInt(uiErrorCode);
		IF NOT arfbAlarm[0].bActive THEN		
			arfbAlarm[0].Raise(nTimeStamp:=0);
		END_IF
	ELSE	
		IF  arfbAlarm[0].bActive AND bReset THEN
			arfbAlarm[0].Clear(nTimeStamp:=0, bResetConfirmation:= FALSE);
		END_IF
// 	udiErrorID													:= 357;//uiErrorCode;
// 	sErrorDescription											:= 'Zresetuj błąd na panelu falownika.';
// 	sErrorDescription2											:= UINT_TO_STRING(uiErrorCode);
END_IF	
 // Alarm_0581	581	Error	Błąd komunikacji z urządzeniem (WcState)                                               	
IF bWcStateError AND bEnable THEN
	IF NOT arfbAlarm[1].bActive THEN		
			arfbAlarm[1].Raise(nTimeStamp:=0);
		END_IF
	ELSE	
		IF  arfbAlarm[1].bActive AND bReset THEN
			arfbAlarm[1].Clear(nTimeStamp:=0, bResetConfirmation:= FALSE);
		END_IF
// 	udiErrorID													:= 358;//INT_TO_UDINT(iIndex + 1) ;	
// 	sErrorDescription											:= 'Błąd komunikacji z urządzeniem (WcState)';
END_IF
// Alarm_0582	582	Error	Utracono gotowość falownika do pracy
IF bLenzeReadinessError AND bEnable THEN
		IF NOT arfbAlarm[2].bActive THEN		
			arfbAlarm[2].Raise(nTimeStamp:=0);
		END_IF
	ELSE	
		IF  arfbAlarm[2].bActive AND bReset THEN
			arfbAlarm[2].Clear(nTimeStamp:=0, bResetConfirmation:= FALSE);
		END_IF
// 	udiErrorID													:= 359;//INT_TO_UDINT(iIndex + 2) ;	
// 	sErrorDescription											:= 'Utracono gotowość falownika do pracy';
END_IF	
// Alarm_0583	583	Error	Przekroczenie czasu oczekiwania na odpowiedź falownika
IF bCheckInitTimeError AND bEnable THEN
		IF NOT arfbAlarm[3].bActive THEN		
			arfbAlarm[3].Raise(nTimeStamp:=0);
		END_IF
	ELSE	
		IF  arfbAlarm[3].bActive AND bReset THEN
			arfbAlarm[3].Clear(nTimeStamp:=0, bResetConfirmation:= FALSE);
		END_IF                             	
// 	udiErrorID													:= 360;//INT_TO_UDINT(iIndex  + 3) ;	
// 	sErrorDescription											:= 'Przekroczenie czasu oczekiwania na odpowiedź falownika';
END_IF	
// Alarm_0584	584	Error	Przepełnienie
IF bFullConveyorError AND bEnable  THEN
	IF NOT arfbAlarm[4].bActive THEN		
			arfbAlarm[4].Raise(nTimeStamp:=0);
		END_IF
	ELSE	
		IF  arfbAlarm[4].bActive AND bReset THEN
			arfbAlarm[4].Clear(nTimeStamp:=0, bResetConfirmation:= FALSE);
		END_IF
// 	udiErrorID													:= 361;//INT_TO_UDINT(iIndex  + 4) ;	
// 	sErrorDescription											:= 'Przepełnienie';
END_IF


	
IF NOT bEnable THEN
	bError														:= FALSE;
	udiErrorID													:= 0;
	sErrorDescription											:= ''; 
END_IF	

(*Wyświetlanie błedu na wyjściu*)
bError							:= FALSE;
FOR nAlarmNumerator := 0 TO 19 DO
	bError						:= bError OR arfbAlarm[nAlarmNumerator].bActive;
END_FOR
	
IF bError THEN

	IF 	eState = E_Station.ePreparingToReady    OR
	    eState = E_Station.eReady               OR      
	    eState = E_Station.eStarting			OR           
	    eState = E_Station.eRunning			    OR  
		eState = E_Station.eStopping			OR    
	   	eState = E_Station.eManualMovement      THEN
		
		eState													:= E_Station.eError;	
	END_IF
                                      
END_IF

IF NOT bError THEN
	udiErrorID													:= 0;
	//sErrorDescription											:= ""; 
	sErrorDescription											:= ''; 
END_IF





sErrorStationName:=WSTRING_TO_STRING(sStationName);
END_ACTION

ACTION ACT_EStop:
IF NOT bEStop THEN
	IF eState <> E_Station.eAborted THEN
		IF eState <> E_Station.eAborting THEN
			eState:= E_Station.eAborting;	
		END_IF
	END_IF
END_IF
END_ACTION

ACTION ACT_ManualMovements:
CASE iManualStep OF
			
	0: (*Oczekiwanie na zbocze narastajace komendy ruchu JOG*)
	
		bEnableOperation										:= bRun;
		
		IF rtJogForward.Q THEN
			tonPressing.IN										:= TRUE;
			tonPressing.PT										:= T#1S;
			iManualStep:= 10;
		END_IF
					
		IF rtJogBackward.Q THEN
			tonPressing.IN										:= TRUE;
			tonPressing.PT										:= T#1S;
			iManualStep:= 20;
		END_IF
		
	
	10: (*Oczekiwanie na zbocze opadajace komendy ruchu JOG w kierunku pozytywnym*)
	
		bEnableOperation												:= TRUE;
	                                                                	
		IF NOT bJogForward THEN	                                    	
			IF tonPressing.Q OR bDeactivateStepMode	THEN            	
				iManualStep:= 100;	
			ELSIF NOT tonPressing.Q AND NOT bDeactivateStepMode THEN	
				tonTimeOfJog.IN											:= TRUE;
				tonTimeOfJog.PT											:= tTimeOfJog;
				iManualStep:= 50;
			END_IF                                                  	
			tonPressing.IN												:= FALSE;
		END_IF
		
	
	20: (*Oczekiwanie na zbocze opadajace komendy ruchu JOG w kierunku negatywnym*)
		
		bEnableOperation												:= TRUE;
	                                                                	
		IF NOT bJogBackward THEN	                                    	
			IF tonPressing.Q OR bDeactivateStepMode	THEN            	
				iManualStep:= 100;	
			ELSIF NOT tonPressing.Q AND NOT bDeactivateStepMode THEN	
				tonTimeOfJog.IN											:= TRUE;
				tonTimeOfJog.PT											:= tTimeOfJog;
				iManualStep:= 50;
			END_IF                                                  	
			tonPressing.IN												:= FALSE;
		END_IF
		
	50: (*Oczekiwanie na odliczenie czasu kroku*)
	
		IF tonTimeOfJog.Q THEN
			tonTimeOfJog.IN												:= FALSE;
			iManualStep:= 100;
		END_IF
		
	100: (*Zakonczenie ruchu*)
	
		bEnableOperation												:= FALSE;
		iManualStep:= 0;	

END_CASE


IF NOT bManualMode THEN
	tonTimeOfJog.IN														:= FALSE;
	tonPressing.IN														:= FALSE;
	bEnableOperation													:= FALSE;
	iManualStep															:= 0;
	eState:= E_Station.eReady;
END_IF
END_ACTION

ACTION ACT_StatusWord:
bReadyToSwitchOn 								:= uiStatusWord.0;
bSwitchedOn 									:= uiStatusWord.1;
bOperationEnabled 								:= uiStatusWord.2;
bFaultActive 									:= uiStatusWord.3;
bVoltageEnabled 								:= uiStatusWord.4; 
bQuickStopActive 								:= uiStatusWord.5; 
bSwitchOnDisabled 								:= uiStatusWord.6;
bWarningActive 									:= uiStatusWord.7; 
bDeactiveRPDOs 									:= uiStatusWord.8; 
bRemote											:= uiStatusWord.9; 
bTargetReached									:= uiStatusWord.10;
bInternalLimitActive							:= uiStatusWord.11;
bReserved6										:= uiStatusWord.12;
bReserved7										:= uiStatusWord.13;
bBreakeReleased									:= uiStatusWord.14;
bSTONotActive									:= uiStatusWord.15;
END_ACTION

ACTION aStationID:
udiStationID	:=	iStationIndex;
END_ACTION

END_FUNCTION_BLOCK

// ---- POUs/P00_Basic.TcPOU
(*
Nazwa:			P00_Basic 
Opis:			Funkcje podstawowe
Wersja:			v0.1
Data:			2018-10-10
Autor:			DP
Urzadzenia:		
Konfiguracja:	
Info:
- Tworzenie zmiennych podstawowych, typu czas, impulsy itd.

*)


PROGRAM P00_Basic
VAR
	fbGetSystemTime			: FB_GetSystemTime;
	fbCycleTimes			: FB_CycleTimes;
	
	Timer1HzOn				: TON;
	Timer1HzOff				: TON;
	Timer2HzOn				: TON;
	Timer2HzOff				: TON;
	
	rtImp1Sec				: R_TRIG;
	
	sDateAndTime			: STRING;
	
END_VAR

a_SystemTime();				// Pobieranie aktualnego czasu
a_CycleTimes();

// Timer 1Hz ##########################
Timer1HzOn (IN := NOT b1Hz, PT := T#1S);
IF Timer1HzOn.Q THEN
	b1Hz := TRUE;
	GVL.bV1Hz := TRUE;
END_IF

Timer1HzOff (IN := b1Hz, PT := T#1S);
IF Timer1HzOff.Q THEN
	b1Hz := FALSE;
	GVL.bV1Hz := FALSE;
END_IF

// Timer 2Hz ##########################
Timer2HzOn (IN := NOT b2Hz, PT := T#500MS);
IF Timer2HzOn.Q THEN
	b2Hz := TRUE;
END_IF

Timer2HzOff (IN := b2Hz, PT := T#500MS);
IF Timer2HzOff.Q THEN
	b2Hz := FALSE;
END_IF

(*Zbocze narastające dla bitu sekundowego*)
rtImp1Sec(CLK := b1Hz , Q=> bImp1Sec);

bAlwaysFalse:=FALSE;

sDateAndTime:= 
Concat(Concat(Concat(Concat(Concat(Concat(Concat(Concat(Concat(Concat(Concat(WORD_TO_STRING(wYear),'-'),WORD_TO_STRING(wMonth)),'-'),WORD_TO_STRING(wDay)),' '),WORD_TO_STRING(wHour)),':'),WORD_TO_STRING(wMinute)),':'),WORD_TO_STRING(wSecond)),';');

ACTION a_CycleTimes:
P02_Dispencers.fbDispencer1.tCycleTime;
P02_Dispencers.fbDispencer2.tCycleTime;
P02_Dispencers.fbDispencerGatesStation.tCycleTime;
P02_Dispencers.fbDispencersCatch1Station.tCycleTime;
P05_Weight.fbWeight1.tCycleTime;
P05_Weight.fbWeight2.tCycleTime;
P05_Weight.fbWeight3.tCycleTime;
P05_Weight.fbWeight4.tCycleTime;
P10_GripperScrewer.fb2GripperScrewer1.tCycleTime;
P10_GripperScrewer.fb2GripperScrewer2.tCycleTime;
P10_GripperScrewer.fbGripperScrewer1CatchStation.tCycleTime;
P13_BottleTransfer.fbBottleTransfer.tCycleTime;




fbCycleTimes(
	bEnable:= TRUE, 
	bReset:= FALSE, 
	tStation1CT:= P02_Dispencers.fbDispencersDragLeftStation.tCycleTime,
	bStation1En:= P02_Dispencers.fbDispencersDragLeftStation.bEnable,
	sStation1Name:= 'Dispencers drag', 
	tStation2CT:= P02_Dispencers.fbDispencer1.tCycleTime, 
	bStation2En:= P02_Dispencers.fbDispencer1.bEnable, 
	sStation2Name:= 'Dispencer 1', 
	tStation3CT:= P02_Dispencers.fbDispencer2.tCycleTime, 
	bStation3En:= P02_Dispencers.fbDispencer2.bEnable, 
	sStation3Name:= 'Dispencer 2', 
	tStation4CT:= P02_Dispencers.fbDispencerGatesStation.tCycleTime, 
	bStation4En:= P02_Dispencers.fbDispencerGatesStation.bEnable, 
	sStation4Name:= 'Dispencers gate', 
	tStation5CT:= P02_Dispencers.fbDispencersCatch1Station.tCycleTime, 
	bStation5En:= P02_Dispencers.fbDispencersCatch1Station.bEnable, 
	sStation5Name:= 'Dispencer catcher', 

	tStation9CT:= P05_Weight.fbWeight1.tCycleTime, 
	bStation9En:= P05_Weight.fbWeight1.bEnable, 
	sStation9Name:= 'Weight 1', 
	
	tStation10CT:= P10_GripperScrewer.fbGripperScrewersDragStation.tCycleTime,
	bStation10En:= P10_GripperScrewer.fbGripperScrewersDragStation.bEnable,
	sStation10Name:= 'Dispencers drag', 	
	
	tStation11CT:= 		P10_GripperScrewer.fb2GripperScrewer1.tCycleTime, 
	bStation11En:= 		P10_GripperScrewer.fb2GripperScrewer1.bEnable1, 
	sStation11Name:= 	'Capping unit 1',  
	
	tStation12CT:= 		P10_GripperScrewer.fb2GripperScrewer2.tCycleTime, 
	bStation12En:= 		P10_GripperScrewer.fb2GripperScrewer2.bEnable1, 
	sStation12Name:= 	'Capping unit 1 2',  
 
	tStation17CT:= 		P10_GripperScrewer.fbGripperScrewer1CatchStation.tCycleTime, 
	bStation17En:= 		P10_GripperScrewer.fbGripperScrewer1CatchStation.bEnable, 
	sStation17Name:= 	'Capping lifter 1',  
	
	tStation17CT:= 		P10_GripperScrewer.fbGripperScrewer2CatchStation.tCycleTime, 
	bStation17En:= 		P10_GripperScrewer.fbGripperScrewer2CatchStation.bEnable, 
	sStation17Name:= 	'Capping lifter 2',  	
	 
	tStation20CT:= 		P13_BottleTransfer.fbBottleTransfer.tCycleTime, 
	bStation20En:= 		P13_BottleTransfer.fbBottleTransfer.bEnable, 
	sStation20Name:= 	'Robot', 	
	sSlowestStation1=> VIS.sSlowestStation1, 
	sSlowestStation2=> VIS.sSlowestStation2, 
	sSlowestStation3=> VIS.sSlowestStation3,
	sSlowestStation4=> ,//VIS.sSlowestStation4,
	sSlowestStation5=> ,//VIS.sSlowestStation5,
	iSlowestStationCount1=> VIS.iSlowestStationCount1,
	iSlowestStationCount2=> VIS.iSlowestStationCount2,	
	iSlowestStationCount3=> VIS.iSlowestStationCount3,
	iSlowestStationCount4=> ,//VIS.iSlowestStationCount4,	
	iSlowestStationCount5=> //VIS.iSlowestStationCount5
	);
END_ACTION

ACTION a_SystemTime:
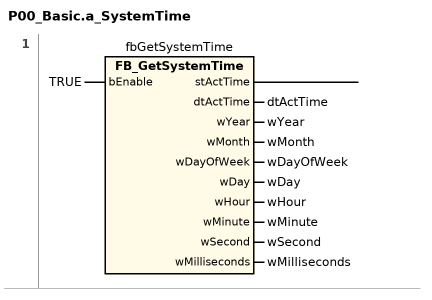
// NETWORK 1
fbGetSystemTime(
    bEnable := TRUE,
    dtActTime => dtActTime,
    wYear => wYear,
    wMonth => wMonth,
    wDayOfWeek => wDayOfWeek,
    wDay => wDay,
    wHour => wHour,
    wMinute => wMinute,
    wSecond => wSecond,
    wMilliseconds => wMilliseconds); // FB_GetSystemTime
END_ACTION

END_PROGRAM

// ---- POUs/FB/DateAndTime/FB_GetSystemTime.TcPOU
(****************************************************************************************)
(*							Beckhoff Automation Poland									*)
(*								FB_GetSystemTime  v1.2									*)
(*									26.07.2013											*)
(*		v1.2 - zmiana nazwy bloku z FB_Time na FB_GetSystemTime, dodanie wyjscia DT		*)
(*		v1.1 - dodano na wyjściu zmienną czasu w formie struktury TIMESTRUCT 			*)
(*				Blok funkcyjny podający dokładną datę w odrębnych zmiennych				*)
(*						może być wywołany raz w programie PLC							*)
(*						Wymaga dodania biblioteki TcUtilities.lib						*)
(*______________________________________________________________________________________*)
FUNCTION_BLOCK FB_GetSystemTime
VAR_INPUT
	bEnable:			BOOL;				(*Aktywuje pobieranie czasu systemowego*)
END_VAR
VAR_OUTPUT
	stActTime			:	TIMESTRUCT;
	dtActTime: DT;
(*Poszczególne składowe daty*)
	wYear 				:	WORD;
	wMonth 				:	WORD;
	wDayOfWeek 			: 	WORD;
	wDay 				:	WORD;
	wHour 				:	WORD;
	wMinute 			:	WORD;
	wSecond 			:	WORD;
	wMilliseconds 		: 	WORD;
END_VAR
VAR
	fbGetTime			:	NT_GetTime;
	Get					:	TON;
END_VAR
VAR CONSTANT
	tFrequency			:	TIME			:= T#1s;				(*Częstotliwość pobierania czasu*)
END_VAR

Get(IN:= NOT Get.Q AND bEnable, PT:=tFrequency);
fbGetTime(
	NETID:= '',
	START:= Get.Q,
	TMOUT:= T#200ms,
	TIMESTR=>stActTime);

dtActTime 		:= SYSTEMTIME_TO_DT(stActTime);
wDay 			:= stActTime.wDay;
wDayOfWeek 		:= stActTime.wDayOfWeek;
wHour 			:= stActTime.wHour;
wMilliseconds 	:= stActTime.wMilliseconds;
wMinute 		:= stActTime.wMinute;
wMonth 			:= stActTime.wMonth;
wSecond 		:= stActTime.wSecond;
wYear 			:= stActTime.wYear;

END_FUNCTION_BLOCK

// ---- POUs/FB/FB_CycleTimes.TcPOU
(*
Nazwa:			FB_CycleTimes
Opis:			czasy cyklów
Wersja:			v0.1
Data:			2019-08-29
Autor:			DP
Urzadzenia:		
Konfiguracja:	
Info: 
- dodano opcje przesuwu liniowego
*)
FUNCTION_BLOCK FB_CycleTimes
VAR_INPUT
	bEnable: BOOL;				//Zezwolenie na pracę
	bReset:BOOL;				//Stop awaryjny nieaktywny
	tStation1CT:TIME;			//Czas cyklu stacji nr 1
	bStation1En:BOOL;			//Zezwolenie pracy stacji nr 1
	sStation1Name:STRING;		//Nazwa stacji nr 1
	tStation2CT:TIME;			//Czas cyklu stacji nr 2
	bStation2En:BOOL;			//Zezwolenie pracy stacji nr 2
	sStation2Name:STRING;		//Nazwa stacji nr 2
	tStation3CT:TIME;			//Czas cyklu stacji nr 3
	bStation3En:BOOL;			//Zezwolenie pracy stacji nr 3
	sStation3Name:STRING;		//Nazwa stacji nr 3
	tStation4CT:TIME;			//Czas cyklu stacji nr 4
	bStation4En:BOOL;			//Zezwolenie pracy stacji nr 4
	sStation4Name:STRING;		//Nazwa stacji nr 4
	tStation5CT:TIME;			//Czas cyklu stacji nr 5
	bStation5En:BOOL;			//Zezwolenie pracy stacji nr 5
	sStation5Name:STRING;		//Nazwa stacji nr 5
	tStation6CT:TIME;			//Czas cyklu stacji nr 6
	bStation6En:BOOL;			//Zezwolenie pracy stacji nr 6
	sStation6Name:STRING;		//Nazwa stacji nr 6
	tStation7CT:TIME;			//Czas cyklu stacji nr 7
	bStation7En:BOOL;			//Zezwolenie pracy stacji nr 7
	sStation7Name:STRING;		//Nazwa stacji nr 7
	tStation8CT:TIME;			//Czas cyklu stacji nr 8
	bStation8En:BOOL;			//Zezwolenie pracy stacji nr 8
	sStation8Name:STRING;		//Nazwa stacji nr 8
	tStation9CT:TIME;			//Czas cyklu stacji nr 9
	bStation9En:BOOL;			//Zezwolenie pracy stacji nr 9
	sStation9Name:STRING;		//Nazwa stacji nr 9
	tStation10CT:TIME;			//Czas cyklu stacji nr 10
	bStation10En:BOOL;			//Zezwolenie pracy stacji nr 10
	sStation10Name:STRING;		//Nazwa stacji nr 10
	tStation11CT:TIME;			//Czas cyklu stacji nr 11
	bStation11En:BOOL;			//Zezwolenie pracy stacji nr 11
	sStation11Name:STRING;		//Nazwa stacji nr 11
	tStation12CT:TIME;			//Czas cyklu stacji nr 12
	bStation12En:BOOL;			//Zezwolenie pracy stacji nr 12
	sStation12Name:STRING;		//Nazwa stacji nr 12
	tStation13CT:TIME;			//Czas cyklu stacji nr 13
	bStation13En:BOOL;			//Zezwolenie pracy stacji nr 13
	sStation13Name:STRING;		//Nazwa stacji nr 13
	tStation14CT:TIME;			//Czas cyklu stacji nr 14
	bStation14En:BOOL;			//Zezwolenie pracy stacji nr 14
	sStation14Name:STRING;		//Nazwa stacji nr 14
	tStation15CT:TIME;			//Czas cyklu stacji nr 15
	bStation15En:BOOL;			//Zezwolenie pracy stacji nr 15	
	sStation15Name:STRING;		//Nazwa stacji nr 15
	tStation16CT:TIME;			//Czas cyklu stacji nr 16
	bStation16En:BOOL;			//Zezwolenie pracy stacji nr 16	
	sStation16Name:STRING;		//Nazwa stacji nr 16
	tStation17CT:TIME;			//Czas cyklu stacji nr 17
	bStation17En:BOOL;			//Zezwolenie pracy stacji nr 17	
	sStation17Name:STRING;		//Nazwa stacji nr 17
	tStation18CT:TIME;			//Czas cyklu stacji nr 18
	bStation18En:BOOL;			//Zezwolenie pracy stacji nr 18	
	sStation18Name:STRING;		//Nazwa stacji nr 18
	tStation19CT:TIME;			//Czas cyklu stacji nr 19
	bStation19En:BOOL;			//Zezwolenie pracy stacji nr 19	
	sStation19Name:STRING;		//Nazwa stacji nr 19
	tStation20CT:TIME;			//Czas cyklu stacji nr 20
	bStation20En:BOOL;			//Zezwolenie pracy stacji nr 20	
	sStation20Name:STRING;		//Nazwa stacji nr 20



	
	
END_VAR
VAR_OUTPUT
	sSlowestStation1:STRING;		//Opis najwolniejszej stacji nr 1
	sSlowestStation2:STRING;		//Opis najwolniejszej stacji nr 2
	sSlowestStation3:STRING;		//Opis najwolniejszej stacji nr 3
	sSlowestStation4:STRING;		//Opis najwolniejszej stacji nr 4
	sSlowestStation5:STRING;		//Opis najwolniejszej stacji nr 5
	iSlowestStationCount1:INT;		//Ilość dla najwolniejszej stacji nr 1	
	iSlowestStationCount2:INT;		//Ilość dla najwolniejszej stacji nr 2		
	iSlowestStationCount3:INT;		//Ilość dla najwolniejszej stacji nr 3	
	iSlowestStationCount4:INT;		//Ilość dla najwolniejszej stacji nr 4		
	iSlowestStationCount5:INT;		//Ilość dla najwolniejszej stacji nr 5		
END_VAR

VAR
	arCycleTimes: ARRAY [1..20] OF S_CycleTimes;
	dTimeTempSlowest1:DINT;
	dTimeTempSlowest2:DINT;
	dTimeTempSlowest3:DINT;
	dTimeTempSlowest4:DINT;
	dTimeTempSlowest5:DINT;
	i: INT;
END_VAR

ErrorHandling();
Cycle();
ManualMovements();
Statistics();

ACTION Cycle:
dTimeTempSlowest1:=0;
dTimeTempSlowest2:=0;
dTimeTempSlowest3:=0;
dTimeTempSlowest4:=0;
dTimeTempSlowest5:=0;


arCycleTimes[1].bEnable:=bStation1En;
arCycleTimes[1].bName:=sStation1Name;
arCycleTimes[1].dTime:=TIME_TO_DINT(tStation1CT);
arCycleTimes[2].bEnable:=bStation2En;
arCycleTimes[2].bName:=sStation2Name;
arCycleTimes[2].dTime:=TIME_TO_DINT(tStation2CT);
arCycleTimes[3].bEnable:=bStation3En;
arCycleTimes[3].bName:=sStation3Name;
arCycleTimes[3].dTime:=TIME_TO_DINT(tStation3CT);
arCycleTimes[4].bEnable:=bStation4En;
arCycleTimes[4].bName:=sStation4Name;
arCycleTimes[4].dTime:=TIME_TO_DINT(tStation4CT);
arCycleTimes[5].bEnable:=bStation5En;
arCycleTimes[5].bName:=sStation5Name;
arCycleTimes[5].dTime:=TIME_TO_DINT(tStation5CT);
arCycleTimes[6].bEnable:=bStation6En;
arCycleTimes[6].bName:=sStation6Name;
arCycleTimes[6].dTime:=TIME_TO_DINT(tStation6CT);
arCycleTimes[7].bEnable:=bStation7En;
arCycleTimes[7].bName:=sStation7Name;
arCycleTimes[7].dTime:=TIME_TO_DINT(tStation7CT);
arCycleTimes[8].bEnable:=bStation8En;
arCycleTimes[8].bName:=sStation8Name;
arCycleTimes[8].dTime:=TIME_TO_DINT(tStation8CT);
arCycleTimes[9].bEnable:=bStation9En;
arCycleTimes[9].bName:=sStation9Name;
arCycleTimes[9].dTime:=TIME_TO_DINT(tStation9CT);
arCycleTimes[10].bEnable:=bStation10En;
arCycleTimes[10].bName:=sStation10Name;
arCycleTimes[10].dTime:=TIME_TO_DINT(tStation10CT);
arCycleTimes[11].bEnable:=bStation11En;
arCycleTimes[11].bName:=sStation11Name;
arCycleTimes[11].dTime:=TIME_TO_DINT(tStation11CT);
arCycleTimes[12].bEnable:=bStation12En;
arCycleTimes[12].bName:=sStation12Name;
arCycleTimes[12].dTime:=TIME_TO_DINT(tStation12CT);
arCycleTimes[13].bEnable:=bStation13En;
arCycleTimes[13].bName:=sStation13Name;
arCycleTimes[13].dTime:=TIME_TO_DINT(tStation13CT);
arCycleTimes[14].bEnable:=bStation14En;
arCycleTimes[14].bName:=sStation14Name;
arCycleTimes[14].dTime:=TIME_TO_DINT(tStation14CT);
arCycleTimes[15].bEnable:=bStation15En;
arCycleTimes[15].bName:=sStation15Name;
arCycleTimes[15].dTime:=TIME_TO_DINT(tStation15CT);
arCycleTimes[16].bEnable:=bStation16En;
arCycleTimes[16].bName:=sStation16Name;
arCycleTimes[16].dTime:=TIME_TO_DINT(tStation16CT);
arCycleTimes[17].bEnable:=bStation17En;
arCycleTimes[17].bName:=sStation17Name;
arCycleTimes[17].dTime:=TIME_TO_DINT(tStation17CT);
arCycleTimes[18].bEnable:=bStation18En;
arCycleTimes[18].bName:=sStation18Name;
arCycleTimes[18].dTime:=TIME_TO_DINT(tStation18CT);
arCycleTimes[19].bEnable:=bStation19En;
arCycleTimes[19].bName:=sStation19Name;
arCycleTimes[19].dTime:=TIME_TO_DINT(tStation19CT);
arCycleTimes[20].bEnable:=bStation20En;
arCycleTimes[20].bName:=sStation20Name;
arCycleTimes[20].dTime:=TIME_TO_DINT(tStation20CT);
//Dodaje na testy


FOR i:=1 TO 20 DO
	IF arCycleTimes[i].bEnable AND arCycleTimes[i].dTime > dTimeTempSlowest1 THEN
		dTimeTempSlowest1:=arCycleTimes[i].dTime;
		//sSlowestStation1:=CONCAT(arCycleTimes[i].bName,CONCAT(':',DINT_TO_STRING(dTimeTempSlowest1))); 
		sSlowestStation1:=arCycleTimes[i].bName;
		iSlowestStationCount1:=DINT_TO_INT(dTimeTempSlowest1);
	END_IF
END_FOR

FOR i:=1 TO 20 DO
	IF arCycleTimes[i].bEnable AND NOT (dTimeTempSlowest1=arCycleTimes[i].dTime) AND arCycleTimes[i].dTime > dTimeTempSlowest2 THEN
		dTimeTempSlowest2:=arCycleTimes[i].dTime;
		//sSlowestStation2:=CONCAT(arCycleTimes[i].bName,CONCAT(':',DINT_TO_STRING(dTimeTempSlowest2))); 
		sSlowestStation2:=arCycleTimes[i].bName;
		iSlowestStationCount2:=DINT_TO_INT(dTimeTempSlowest2);
	END_IF
END_FOR
	

FOR i:=1 TO 20 DO
	IF arCycleTimes[i].bEnable AND NOT (dTimeTempSlowest1=arCycleTimes[i].dTime) AND NOT (dTimeTempSlowest2=arCycleTimes[i].dTime) AND arCycleTimes[i].dTime > dTimeTempSlowest3 THEN
		dTimeTempSlowest3:=arCycleTimes[i].dTime;
		//sSlowestStation3:=CONCAT(arCycleTimes[i].bName,CONCAT(':',DINT_TO_STRING(dTimeTempSlowest3))); 
		sSlowestStation3:=arCycleTimes[i].bName;
		iSlowestStationCount3:=DINT_TO_INT(dTimeTempSlowest3);
	END_IF
END_FOR

FOR i:=1 TO 20 DO
	IF arCycleTimes[i].bEnable AND NOT (dTimeTempSlowest1=arCycleTimes[i].dTime) AND NOT (dTimeTempSlowest2=arCycleTimes[i].dTime) AND NOT (dTimeTempSlowest3=arCycleTimes[i].dTime) AND arCycleTimes[i].dTime > dTimeTempSlowest4 THEN
		dTimeTempSlowest4:=arCycleTimes[i].dTime;
		//sSlowestStation4:=CONCAT(arCycleTimes[i].bName,CONCAT(':',DINT_TO_STRING(dTimeTempSlowest4))); 
		sSlowestStation4:=arCycleTimes[i].bName;
		iSlowestStationCount4:=DINT_TO_INT(dTimeTempSlowest4);
	END_IF
END_FOR

FOR i:=1 TO 20 DO
	IF arCycleTimes[i].bEnable AND NOT (dTimeTempSlowest1=arCycleTimes[i].dTime) AND NOT (dTimeTempSlowest2=arCycleTimes[i].dTime) AND NOT (dTimeTempSlowest3=arCycleTimes[i].dTime) AND NOT (dTimeTempSlowest4=arCycleTimes[i].dTime) AND arCycleTimes[i].dTime > dTimeTempSlowest5 THEN
		dTimeTempSlowest5:=arCycleTimes[i].dTime;
		//sSlowestStation5:=CONCAT(arCycleTimes[i].bName,CONCAT(':',DINT_TO_STRING(dTimeTempSlowest5))); 
		sSlowestStation5:=arCycleTimes[i].bName;
		iSlowestStationCount5:=DINT_TO_INT(dTimeTempSlowest5);
	END_IF
END_FOR
END_ACTION

ACTION ErrorHandling:

END_ACTION

ACTION ManualMovements:

END_ACTION

ACTION Statistics:

END_ACTION

END_FUNCTION_BLOCK

// ---- POUs/P00_Counters.TcPOU
(*
Nazwa:			P00_Counters 
Opis:			Liczenie formatek
Wersja:			v0.1
Data:			2018-10-10
Autor:			DP
Urzadzenia:		
Konfiguracja:	
Info:
- wydajności chwilowe, sumaryczne na podstawie czasu pracy lini

*)
PROGRAM P00_Counters
VAR
	fbCountersLog											: FB_SaveLineToFile;	

	tonMinuteTimer											: TON;
	tonMinuteTicksWhenCycleOn								: TON;
	tonMachineCycleTimer									: TON;
	
	rtSaveCounters											: R_TRIG;
	RtMachineCycleTimerRead									: R_TRIG;
	
	nMinuteCount											: UDINT;		// licznik minut
	udiGlobalCounterTemp									: UDINT;
	
	uiWheelBottlesCounter									: UINT;
	nShiftBottlesCounterAux									: UINT;
	
	btestint												: INT;
	
	bCountersLogBusy										: BOOL;
	bCountersLogError										: BOOL;

	tMachineCycleTimeTemp: TIME;
		
	
	fbGlobalCounterSave										: FB_SaveTextToFile;	
	fbGlobalCounterRead										: FB_ReadTextFromFile;	
	rtLoadCounters: R_TRIG;
	tfBusy: F_TRig;
	uiCounterShiftBottlesTemp 								:UINT;
    uiCounterShiftBottlesLast   							:UINT; 
	AuiCounterInstantEfficiencyLast							:ARRAY [1..10] OF  UINT; // Wydajność chwilowa prawidłowych butelek [szt./h]	 
	ftIbFirstFormCheckFormSensor							:F_TRIG;
	
	//Wydajność wersja 2
	udiEfficiencyCycleTime									:	UDINT;
	tEfficiencyStartTime									:	TIME;
	lrEfficiencyCycleTimeSum								:	LREAL;
	lrEffectivicyAverage									:	LREAL;		
	tonEfficiencyMachineWorking								:	TON;
	rtEfficiencyOutSensor									:	R_TRIG;
	fbEfficiencyOutSensor									:	FB_InputFilter_V2;
	AudiEfficiencyCycleTime									:	ARRAY [0..iEfficiencyAverageBuferSize-1] OF LREAL;
	tofEfficiencyOutAndNoBottle								:	TOF;
	bEfficiencyOutAndBottle									:	BOOL;
	rtEfficiencyOutAndNoBottle								:	R_TRIG;
	irtEfficiencyOutAndNoBottle								:	INT;
	//Koniec Wydajność wersja 2
	
	//Wydajność wersja 3
	
	AbEfficiencyBottle											: ARRAY [1..300] OF BOOL;	
	tonEfficiencyBottleMachineWorking							: TON;
	udiEfficiencyBottleSum										: UDINT;
	iEfficincyBottle											: INT;
	bEfficincyBottleTrig										: BOOL;
	//Koniec Wydajność wersja 3	
	
END_VAR
VAR CONSTANT
	iEfficiencyAverageBuferSize									:	INT:=20;
END_VAR

(*Resetowanie licznika*)
IF P00_PackML.fbPMLAuto.ePMLState = E_PMLState.ePMLState_STARTING THEN
	nShiftBottlesCounterAux := 0;
	uiWheelBottlesCounter	:=	0;
END_IF

sCountersToFile();

aEfficiencyBottle();
//DO sprawdzenia

tonMinuteTimer(IN:=(NOT tonMinuteTimer.Q AND NOT VIS.bCounterReset),PT:=T#20S);
tonMinuteTimer.ET;

IF tonMinuteTimer.Q THEN
	nMinuteCount:=nMinuteCount+1;
	VIS.uiCounterAverageEfficiency:=UDINT_TO_UINT(VIS.udiCounterShiftBottles/nMinuteCount)*180;
END_IF

ftIbFirstFormCheckFormSensor(CLK:=P13_BottleTransfer.IbFirstFormCheckFormSensor,Q=>);
// Ziczanie drugim na testy na 30s
IF ftIbFirstFormCheckFormSensor.Q THEN	
	nShiftBottlesCounterAux	:= nShiftBottlesCounterAux + 1;
END_IF

// Wydajność formatek
tonMinuteTicksWhenCycleOn(IN:=((P00_PackML.fbPMLAuto.ePMLState = E_PMLState.ePMLState_EXECUTE ) OR (P00_PackML.fbPMLAuto.ePMLState = E_PMLState.ePMLState_COMPLETING) OR (P00_PackML.fbPMLAuto.ePMLState = E_PMLState.ePMLState_STOPPING)) AND NOT
tonMinuteTicksWhenCycleOn.Q AND NOT VIS.bCounterReset,PT:=T#30S);
IF tonMinuteTicksWhenCycleOn.Q THEN
	VIS.uiCounterMachineEfficiency:=(nShiftBottlesCounterAux*120)/60;
	IF VIS.uiCounterMachineEfficiency > 30 AND VIS.uiCounterMachineEfficiency < 60 THEN
		VIS.uiCounterMachineEfficiency	:=	VIS.uiCounterMachineEfficiency + REAL_TO_UINT(VIS.uiCounterMachineEfficiency*0.02);
	END_IF		
	nShiftBottlesCounterAux:=0;
END_IF
///////


(*Czas cyklu maszyny*)
VIS.udiCounterGlobal;
tonMachineCycleTimer(IN:= VIS.udiCounterGlobal=udiGlobalCounterTemp,PT:=T#1D);
IF tonMachineCycleTimer.IN THEN (*Przepisywanie wartości do zmiennej tymczasowej*)
tMachineCycleTimeTemp:=tonMachineCycleTimer.ET;
END_IF
rtMachineCycleTimerRead(CLK:=(VIS.udiCounterGlobal>udiGlobalCounterTemp));
IF rtMachineCycleTimerRead.Q THEN
	IF tMachineCycleTimeTemp < T#10S THEN // Wpisuj tylko jak mniejsze
		tMachineCycleTime:=tMachineCycleTimeTemp;
	END_IF
	btestint:=btestint+1;
	udiGlobalCounterTemp := VIS.udiCounterGlobal;	
END_IF


//Kasowanie liczników 
IF 	VIS.bCounterReset THEN
	
	VIS.nDialogBoxType	:=	3;														//Wyświetlanie przycisku OK i Anyluj
	VIS.bDialogBoxText	:=	'Are you sure you want to reset the counters?';
	VIS.sDialogBoxPicture	:= 'info';
	VIS.bDialogBoxOn	:=	TRUE;
	
	IF VIS.bDialogBoxAck THEN	
		VIS.bBadPackageReasonReset := TRUE;
		nMinuteCount:=0;
		VIS.uiCounterAverageEfficiency:=0;
		VIS.udiCounterShiftBottles:=0;
		VIS.uiCounterInstantEfficiency:=0;
		nShiftBottlesCounterAux := 0;
		VIS.uiCounterGoodBottles:=0;
		VIS.uiCounterBadBottles:=0;
		VIS.bCounterReset:=FALSE;	
		udiCounterExecuteTimeTemp:=0;	
		udiCounterReadyTimeTemp:=0;	
		udiCounterErrorTimeTemp:=0;	
		VIS.udiCounterExecuteTime:=0;
		VIS.udiCounterReadyTime:=0;	
		VIS.udiCounterErrorTime:=0;	
		VIS.udiCounterGlobalBadBottles:=0;
		uiCounterShiftBottlesLast:=0;
		P00_Visualization.aResetDialog();	
	ELSIF VIS.bDialogBoxCancelAck THEN
		VIS.bCounterReset:=FALSE;
		P00_Visualization.aResetDialog();	
	END_IF
	
END_IF

VIS.udiCounterGlobal; //PODGLĄD LICZNIKA GLOBALNEGO


















































//Jedna butelka dobra:  
//P13_BottleTransfer.fbBottleTransfer.eRunningState>ePicking AND P00_PackML.aP13_BottleTransfer.iRobotPickCase=100 THEN

 //Dwie butelki dobre:
//P13_BottleTransfer.fbBottleTransfer.eRunningState>ePicking AND P00_PackML.aP13_BottleTransfer.iRobotPickCase=200 THEN
(*
ton100msSampleTimer(IN := NOT ton100msSampleTimer.Q, PT := T#100MS);

usiBottleCountInSample := 0;

IF P13_BottleTransfer.fbBottleTransfer.eRunningState > ePicking THEN
    IF P00_PackML.iRobotPickCase <> usiLastPickCase THEN
        IF P00_PackML.iRobotPickCase =100 THEN
            usiBottleCountInSample := 1;
		ELSIF P00_PackML.iRobotPickCase =200 THEN
            usiBottleCountInSample := 2;
        END_IF
        usiLastPickCase :=INT_TO_USINT( P00_PackML.iRobotPickCase );
    END_IF
END_IF

IF bFirstScan OR VIS.bCounterReset THEN
    bFirstScan := FALSE;
    FOR i := 0 TO 1199 DO
        aEfficiencyArray[i] := 0;
    END_FOR
    iSampleIndex := 0;
    udiQuanOfBottleinBuff := 0;
    udiEfficiencyBPM := 0;
END_IF

IF ton100msSampleTimer.Q THEN
    ton100msSampleTimer(IN := FALSE);

    udiQuanOfBottleinBuff := udiQuanOfBottleinBuff - aEfficiencyArray[iSampleIndex];
    aEfficiencyArray[iSampleIndex] := usiBottleCountInSample;
    udiQuanOfBottleinBuff := udiQuanOfBottleinBuff + usiBottleCountInSample;

    iSampleIndex := (iSampleIndex + 1) MOD 1200;

    udiEfficiencyBPM := udiQuanOfBottleinBuff / 2;
END_IF*)

ACTION aEfficiencyBottle:
fbEfficiencyOutSensor(bIn:=P16_LabelMachine.IbLabelMachineFullSensor,	tFilterTimeOn:=T#50MS, tFilterTimeOff:=T#50MS);
rtEfficiencyOutSensor(CLK:=fbEfficiencyOutSensor.bOut, Q=>);

tonEfficiencyBottleMachineWorking(IN:= NOT tonEfficiencyBottleMachineWorking.Q,PT:=T#200MS);


IF rtEfficiencyOutSensor.Q AND 
	(
	(P00_PackML.fbPMLAuto.ePMLState = Tc3_PackML.E_PMLState.ePMLState_STARTING) OR
	(P00_PackML.fbPMLAuto.ePMLState = Tc3_PackML.E_PMLState.ePMLState_EXECUTE) OR 
	(P00_PackML.fbPMLAuto.ePMLState = Tc3_PackML.E_PMLState.ePMLState_STOPPING) 
	) 
THEN // Przeniesione liczenie z robota
	//VIS.uiCounterGoodBottles										:=	VIS.uiCounterGoodBottles+1;
	//VIS.udiCounterGlobal											:=	VIS.udiCounterGlobal+1;
	//VIS.udiCounterShiftBottles										:=	VIS.udiCounterShiftBottles+1;
END_IF	
					
IF tonEfficiencyBottleMachineWorking.Q THEN
	IF 
		(P00_PackML.fbPMLAuto.ePMLState = Tc3_PackML.E_PMLState.ePMLState_STARTING) OR
		(P00_PackML.fbPMLAuto.ePMLState = Tc3_PackML.E_PMLState.ePMLState_EXECUTE) OR 
		(P00_PackML.fbPMLAuto.ePMLState = Tc3_PackML.E_PMLState.ePMLState_STOPPING)  
		THEN
			
			FOR i:=300 TO 2 BY - 1 DO		
				AbEfficiencyBottle[i]	:=	AbEfficiencyBottle[i-1];	
			END_FOR 	
			AbEfficiencyBottle[1]	:=	P16_LabelMachine.IbLabelMachineFullSensor AND NOT bEfficincyBottleTrig;
			
			IF P16_LabelMachine.IbLabelMachineFullSensor THEN
				bEfficincyBottleTrig	:= TRUE;
			END_IF
			IF 	NOT P16_LabelMachine.IbLabelMachineFullSensor THEN
				bEfficincyBottleTrig	:= FALSE;
			END_IF
		
			udiEfficiencyBottleSum	:=	 0;
			FOR i:=1 TO 300 DO	
				udiEfficiencyBottleSum	:=	udiEfficiencyBottleSum + BOOL_TO_UDINT(AbEfficiencyBottle[i]);	
			END_FOR 	
			lrEffectivicyAverage			:=UDINT_TO_LREAL(udiEfficiencyBottleSum);
	ELSE
			FOR i:=1 TO 300 DO	
				AbEfficiencyBottle[i]	:= 0;
			END_FOR 		
		
			udiEfficiencyBottleSum		:=	0;			
			lrEffectivicyAverage		:=	UDINT_TO_LREAL(udiEfficiencyBottleSum);
	END_IF	
END_IF

IF lrEffectivicyAverage	> VIS.uiCounterMachineEfficiency THEN
	lrEffectivicyAverage := VIS.uiCounterMachineEfficiency;
END_IF
VIS.uiCounterInstantEfficiency	:=	LREAL_TO_UINT(lrEffectivicyAverage);
 //Zabezpieczenie przed wartością większą niż maszyny
END_ACTION

ACTION sCountersToFile:
(*
Nazwa:			sCountersToFile
Opis:			Zapisywanie danych do pliku
Wersja:			v0.1
Data:			2019-08-05
Autor:			DP
Urzadzenia:		
Konfiguracja:	
Info:
- zapisywanie do pliku licznika globalnego raz na 10000 formatek, na wszelki wypadek
jakby presistenty znikneły
- wydajności globalne, chwilowe i średnie
*)

VIS.udiCounterGlobal;									//Licznik globalny
VIS.uiCounterInstantEfficiency; 			(**)		//Wydajnoć chwilowa maszyny [szt/h]
VIS.uiCounterAverageEfficiency;			(**)		//Średnia wydajnoć Konfekcji [szt/h]
	
(*Wyznaczanie impulsu do zapisu licznika*)
rtSaveCounters(CLK:=VIS.udiCounterGlobal > nGlobalCounterTemp + 10000, Q=>);
IF rtSaveCounters.Q THEN
	nGlobalCounterTemp := VIS.udiCounterGlobal;
END_IF

rtLoadCounters(CLK:=VIS.udiCounterGlobal=0, Q=>);

(*ZAPISYWANIE LICZNIKÓW DO PLIKU*)
fbCountersLog(
	bExecute:= rtSaveCounters.Q,
	AmsNetId:= , 
	sPath:='C:\Logi\', 
	sName:= 'Liczniki.txt', 
	sLine:= Concat('$R$N',Concat(P00_Basic.sDateAndTime,Concat(Concat(Concat(Concat(UDINT_TO_STRING(VIS.udiCounterGlobal),';'),UDINT_TO_STRING(VIS.uiCounterInstantEfficiency)),';'),UDINT_TO_STRING(VIS.uiCounterAverageEfficiency)))),	 
	bBusy=>bCountersLogBusy , 
	bError=> bCountersLogError);

fbGlobalCounterSave(
	bExecute:= rtSaveCounters.Q,
	AmsNetId:= , 
	sPath:='C:\Logi\', 
	sName:= 'ActualLicznik.txt', 
	sLine:= UDINT_TO_STRING(VIS.udiCounterGlobal),	 
	bBusy=> , 
	bError=> );

fbGlobalCounterRead(
	bExecute:= rtLoadCounters.Q,
	AmsNetId:= , 
	sPath:='C:\Logi\', 
	sName:= 'ActualLicznik.txt', 
	sLine	=> ,	 
	bBusy	=> , 
	bError	=> );
	
tfBusy(Clk:= fbGlobalCounterRead.bBusy);
	
	IF tfBusy.Q AND NOT fbGlobalCounterRead.bError THEN
		VIS.udiCounterGlobal := STRING_TO_UDINT(fbGlobalCounterRead.sLine); 		
	END_IF
END_ACTION

END_PROGRAM

// ---- POUs/FB/FileAccess/FB_SaveLineToFile.TcPOU
(****************************************************************************************)
(*							Beckhoff Automation Poland									*)
(*								FB_SaveLineToFile  v2.0									*)
(*									26.06.2014											*)
(*						Blok funkcyjny zapisujacy tekst do pliku						*)
(*______________________________________________________________________________________
	Versions:
		v1.1	05.08.2016	* Przepisana wersja do TwinCat3
		v1.0	17.09.2012	* Podstawowa wersja z TwinCat2
________________________________________________________________________________________*)
FUNCTION_BLOCK FB_SaveLineToFile
VAR_INPUT
	bExecute	: BOOL;			(* Komenda wpisu *)
	AmsNetId	: T_AmsNetId;	(* AMS NET ID obiektu docelowego, gdy lokalnie, to zmienna moze byc pusta *)
	sPath		: STRING; 		(* Sciezka pliku, np  'Hard Disk\'*)
	sName		: STRING; 		(* Nazwa pliku wraz z rozszerzeniem 'LogFile.txt'; *)
	sLine		: STRING;		(* Tresc wpisu *)
END_VAR
VAR_OUTPUT
	bBusy		: BOOL;
	bError		: BOOL;
END_VAR
VAR
	fbFileOpen	: FB_FileOpen;
	ftOpen		: F_TRIG;
	fbFilePuts	: FB_FilePuts;
	ftPuts		: F_TRIG;
	fbFileClose	: FB_FileClose;
	ftClose		: F_TRIG;
END_VAR
VAR // added by the converter: edge detectors and wires of the graphical bodies
    _w1 : BOOL;
END_VAR

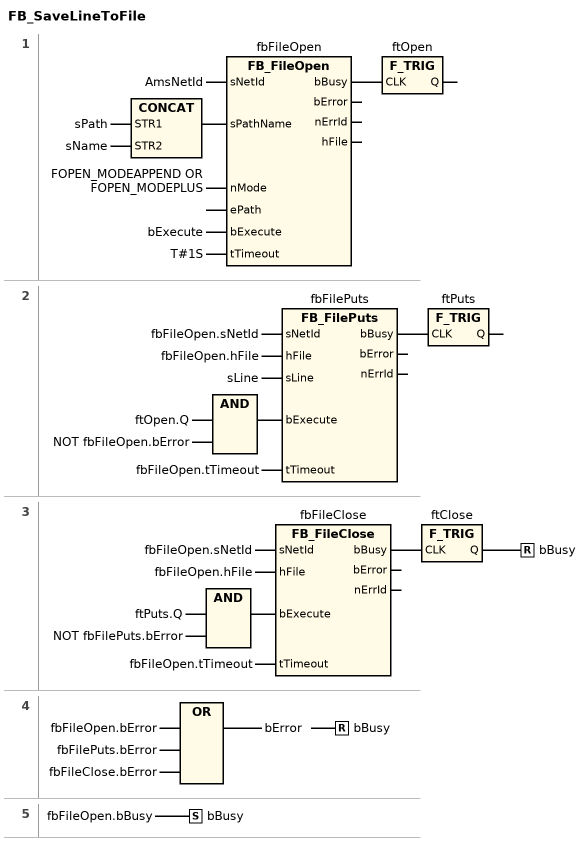
// NETWORK 1
fbFileOpen(
    sNetId := AmsNetId,
    sPathName := CONCAT(STR1 := sPath, STR2 := sName),
    nMode := FOPEN_MODEAPPEND OR FOPEN_MODEPLUS,
    bExecute := bExecute,
    tTimeout := T#1S); // FB_FileOpen
ftOpen(CLK := fbFileOpen.bBusy); // F_TRIG

// NETWORK 2
fbFilePuts(
    sNetId := fbFileOpen.sNetId,
    hFile := fbFileOpen.hFile,
    sLine := sLine,
    bExecute := ftOpen.Q AND (NOT fbFileOpen.bError),
    tTimeout := fbFileOpen.tTimeout); // FB_FilePuts
ftPuts(CLK := fbFilePuts.bBusy); // F_TRIG

// NETWORK 3
fbFileClose(
    sNetId := fbFileOpen.sNetId,
    hFile := fbFileOpen.hFile,
    bExecute := ftPuts.Q AND (NOT fbFilePuts.bError),
    tTimeout := fbFileOpen.tTimeout); // FB_FileClose
ftClose(CLK := fbFileClose.bBusy); // F_TRIG
bBusy R= ftClose.Q;

// NETWORK 4
_w1 := fbFileOpen.bError OR fbFilePuts.bError OR fbFileClose.bError;
bError := _w1;
bBusy R= _w1;

// NETWORK 5
bBusy S= fbFileOpen.bBusy;

END_FUNCTION_BLOCK

// ---- POUs/FB/FileAccess/FB_SaveTextToFile.TcPOU
(****************************************************************************************)
(*							Beckhoff Automation Poland									*)
(*								FB_SaveLineToFile  v2.0									*)
(*									26.06.2014											*)
(*						Blok funkcyjny zapisujacy tekst do pliku						*)
(*______________________________________________________________________________________
	Versions:
		v1.1	05.08.2016	* Przepisana wersja do TwinCat3
		v1.0	17.09.2012	* Podstawowa wersja z TwinCat2
________________________________________________________________________________________*)
FUNCTION_BLOCK FB_SaveTextToFile
VAR_INPUT
	bExecute		: BOOL;			(* Komenda wpisu *)
	AmsNetId		: T_AmsNetId;	(* AMS NET ID obiektu docelowego, gdy lokalnie, to zmienna moze byc pusta *)
	sPath			: STRING; 		(* Sciezka pliku, np  'Hard Disk\'*)
	sName			: STRING; 		(* Nazwa pliku wraz z rozszerzeniem 'LogFile.txt'; *)
	sLine			: STRING;		(* Tresc wpisu *)
END_VAR

VAR_OUTPUT
	bBusy		: BOOL;
	bError		: BOOL;
END_VAR
VAR
	fbFileOpen	: FB_FileOpen;
	ftOpen		: F_TRIG;
	fbFilePuts	: FB_FilePuts;
	ftPuts		: F_TRIG;
	fbFileClose	: FB_FileClose;
	ftClose		: F_TRIG;
END_VAR
VAR // added by the converter: edge detectors and wires of the graphical bodies
    _w1 : BOOL;
END_VAR

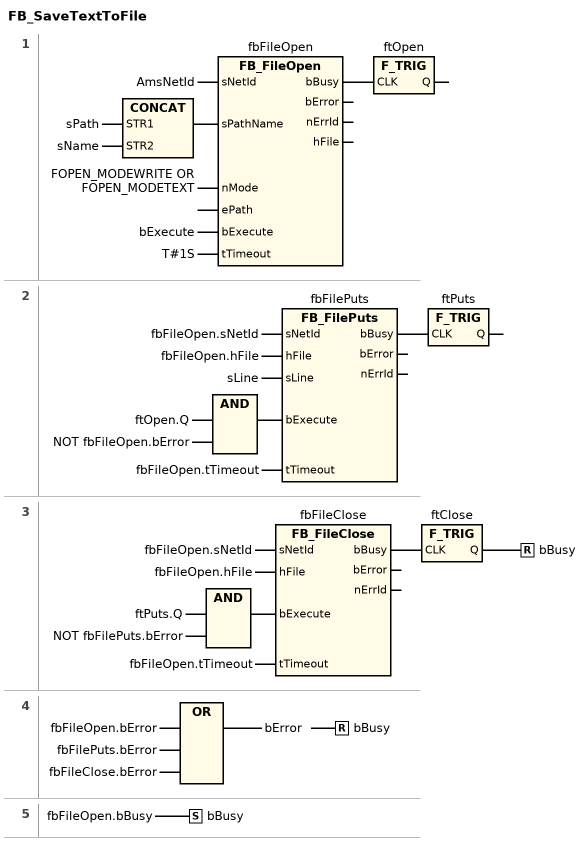
// NETWORK 1
fbFileOpen(
    sNetId := AmsNetId,
    sPathName := CONCAT(STR1 := sPath, STR2 := sName),
    nMode := FOPEN_MODEWRITE OR FOPEN_MODETEXT,
    bExecute := bExecute,
    tTimeout := T#1S); // FB_FileOpen
ftOpen(CLK := fbFileOpen.bBusy); // F_TRIG

// NETWORK 2
fbFilePuts(
    sNetId := fbFileOpen.sNetId,
    hFile := fbFileOpen.hFile,
    sLine := sLine,
    bExecute := ftOpen.Q AND (NOT fbFileOpen.bError),
    tTimeout := fbFileOpen.tTimeout); // FB_FilePuts
ftPuts(CLK := fbFilePuts.bBusy); // F_TRIG

// NETWORK 3
fbFileClose(
    sNetId := fbFileOpen.sNetId,
    hFile := fbFileOpen.hFile,
    bExecute := ftPuts.Q AND (NOT fbFilePuts.bError),
    tTimeout := fbFileOpen.tTimeout); // FB_FileClose
ftClose(CLK := fbFileClose.bBusy); // F_TRIG
bBusy R= ftClose.Q;

// NETWORK 4
_w1 := fbFileOpen.bError OR fbFilePuts.bError OR fbFileClose.bError;
bError := _w1;
bBusy R= _w1;

// NETWORK 5
bBusy S= fbFileOpen.bBusy;

END_FUNCTION_BLOCK

// ---- POUs/FB/FileAccess/FB_ReadTextFromFile.TcPOU
FUNCTION_BLOCK FB_ReadTextFromFile
VAR_INPUT
	bExecute		: BOOL;			(* Komenda odczytu *)
	AmsNetId		: T_AmsNetId;	(* AMS NET ID obiektu docelowego, gdy lokalnie, to zmienna moze byc pusta *)
	sPath			: STRING; 		(* Sciezka pliku, np  'Hard Disk\'*)
	sName			: STRING; 		(* Nazwa pliku wraz z rozszerzeniem 'LogFile.txt'; *)
END_VAR

VAR_OUTPUT
	bBusy		: BOOL;
	bError		: BOOL;
	sLine		: STRING;		(* Tresc wpisu *)
END_VAR
VAR
	fbFileOpen	: FB_FileOpen;
	ftOpen		: F_TRIG;
	fbFileGets	: FB_FileGets;
	ftGets		: F_TRIG;
	fbFileClose	: FB_FileClose;
	ftClose		: F_TRIG;
END_VAR
VAR // added by the converter: edge detectors and wires of the graphical bodies
    _w1 : BOOL;
END_VAR

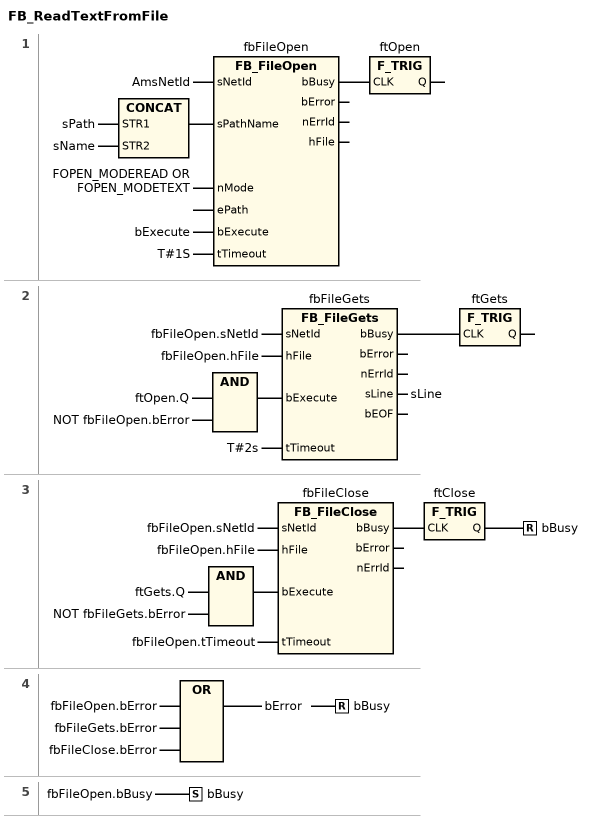
// NETWORK 1
fbFileOpen(
    sNetId := AmsNetId,
    sPathName := CONCAT(STR1 := sPath, STR2 := sName),
    nMode := FOPEN_MODEREAD OR FOPEN_MODETEXT,
    bExecute := bExecute,
    tTimeout := T#1S); // FB_FileOpen
ftOpen(CLK := fbFileOpen.bBusy); // F_TRIG

// NETWORK 2
fbFileGets(
    sNetId := fbFileOpen.sNetId,
    hFile := fbFileOpen.hFile,
    bExecute := ftOpen.Q AND (NOT fbFileOpen.bError),
    tTimeout := T#2s,
    sLine => sLine); // FB_FileGets
ftGets(CLK := fbFileGets.bBusy); // F_TRIG

// NETWORK 3
fbFileClose(
    sNetId := fbFileOpen.sNetId,
    hFile := fbFileOpen.hFile,
    bExecute := ftGets.Q AND (NOT fbFileGets.bError),
    tTimeout := fbFileOpen.tTimeout); // FB_FileClose
ftClose(CLK := fbFileClose.bBusy); // F_TRIG
bBusy R= ftClose.Q;

// NETWORK 4
_w1 := fbFileOpen.bError OR fbFileGets.bError OR fbFileClose.bError;
bError := _w1;
bBusy R= _w1;

// NETWORK 5
bBusy S= fbFileOpen.bBusy;

END_FUNCTION_BLOCK

// ---- POUs/P00_Persistent.TcPOU
(*
Nazwa:			P00_FlowMeters
Opis:			Przepływ powietrza
Wersja:			v0.1
Data:			2018-10-10
Autor:			DP
Urzadzenia:		
Konfiguracja:	
Info:

*)
PROGRAM P00_Persistent
VAR
	fbPersistent:				FB_Persistent;
	bParametersChanged			: BOOL;
	
	bBusy						: BOOL;
	bErr						: BOOL;
	udErrid						: UDINT;
END_VAR

a_Persistent();

//zapisanie zmiennych Persistent, gdy zmiana wartości parametrów lub maszyna wyłączana (brak napięcia zasilania)
bParametersChanged := FALSE;

ACTION a_Persistent:
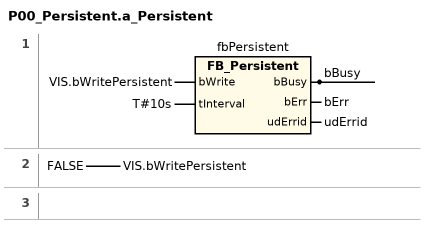
// NETWORK 1
fbPersistent(
    bWrite := VIS.bWritePersistent,
    tInterval := T#10s,
    bBusy => bBusy,
    bErr => bErr,
    udErrid => udErrid); // FB_Persistent

// NETWORK 2
VIS.bWritePersistent := FALSE;

// NETWORK 3
END_ACTION

END_PROGRAM

// ---- POUs/FB/Various/FB_Persistent.TcPOU
FUNCTION_BLOCK FB_Persistent

(********************************************************************************************************)
(*								Beckhoff Automation Poland												*)
(* 									FB_Persistent 	v1.5												*)
(* 										20.08.2014														*)
(* 							v1.5 - zmiana minimalnego interwalu zapisu									*)
(* 					Blok funkcyjny zapisujący zmienne typu persistent na karcie CF						*)
(* 						Możliwy zapis na żądanie lub z określoną częstotliwością.  						*)
(* 				Pozostawienie wejscia tInterval bez zmiennej wyłacza funkcję zapisu cyklicznego			*)
(* 							Minimalny czas między zapisem cyklicznym 30s								*)
(* 				Konieczne jest dodanie biblioteki TcUtilities.lib, TcSystem.lib oraz TcBase.lib			*)
(*			 UWAGA: Blok przygotowany dla RunTime 1 port 801 - typowa konfiguracja 						*)
(*______________________________________________________________________________________________________*)

VAR_INPUT
	bWrite					: BOOL;						(*Zapis na rozkaz *)
	tInterval				: TIME:=T#71582M47S295MS;	(*Czestotliwosc zapisu na karte CF*)
END_VAR
VAR_OUTPUT
	bBusy					: BOOL;
	bErr					: BOOL;
	udErrID					: UDINT;
END_VAR
VAR
	fbWritePersistentData	: FB_WritePersistentData; 	(* Blok zapisu *)
	t1						: TON;						(* Timer zapisu *)
	_GETCURTASKINDEX		: GETCURTASKINDEX;			(* Informacja o Tasku *)
	BIndex					: BYTE;						(* Nr tasku *)
END_VAR

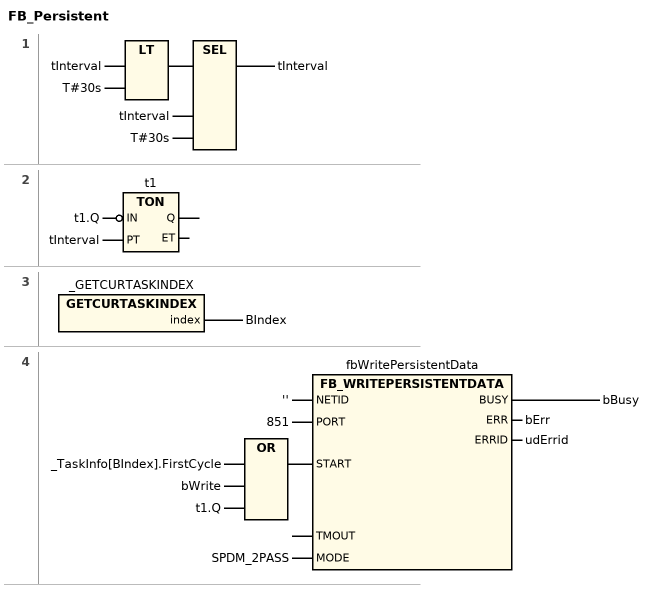
// NETWORK 1
tInterval := SEL(tInterval < T#30s, tInterval, T#30s);

// NETWORK 2
t1(IN := NOT t1.Q, PT := tInterval); // TON

// NETWORK 3
_GETCURTASKINDEX(); // GETCURTASKINDEX
BIndex := _GETCURTASKINDEX.index;

// NETWORK 4
fbWritePersistentData(
    NETID := '',
    PORT := 851,
    START := _TaskInfo[BIndex].FirstCycle OR bWrite OR t1.Q,
    MODE := SPDM_2PASS,
    ERR => bErr,
    ERRID => udErrid); // FB_WRITEPERSISTENTDATA
bBusy := fbWritePersistentData.BUSY;

END_FUNCTION_BLOCK

// ---- POUs/P00_OEE.TcPOU
PROGRAM P00_OEE
VAR
	//Czasy cyklu 
	fbOEECycleTimes							: FB_OEECycleTimes;
	//Powody odrzuceń           			
	fbOEERejectionReason1					: FB_OEERejectionReason;
	fbOEERejectionReason2					: FB_OEERejectionReason;
	//Przezbrajanie             			
	fbMachinePartsChangeover				: FB_InputFilter;
	
	rtChangeover							: R_TRIG;
	rtfbOEERejectionReason2bDone			: R_TRIG;
	
	sOEERejectionReason1Temp				: STRING;
	sOEERejectionReason2Temp				: STRING;
	
	ifbOEERejectionReason2bAddReasonCount	: INT;
	ifbOEERejectionReason1bAddReasonCount	: INT;
	irtfbOEERejectionReason2bDoneCount		: INT;
	rtfbOEERejectionReason1bDone: R_TRIG;
	irtfbOEERejectionReason1bDoneCount: INT;
	rtORRAdd1sec: R_TRIG;
	tofIbBottleInFormCheckBottleSensor : TOF;

	fbOEERaportLog							: FB_SaveLineToFile;	
	rtOEERaportLogAddLine					: R_TRIG;
	wOEERaportMinuteTemp					: WORD;

	fbOEERaportRejectionLog					: FB_SaveLineToFile;	
	sOEEDateAndTime							: STRING;
	sOEEFileDateAndTime						: STRING;
	sOEEFRejectionLine						: STRING;
	rtOEERaportChooseRecipe					: R_TRIG;	
	bOEETest1								: BOOL;
	tonbOEEGenRaport						: TON;
	sOEEActiveErrorIDs						: STRING;
END_VAR

aCycleTimes();
aRejectionReason();
aMachinePartsChangeover();
aOEETime();
aOEERaport();
aOEEPackMLSuspendedReason();

ACTION aCycleTimes:


tMachineCycleTime;

P02_Dispencers.fbDispencersDragRightStation.tCycleTime;
P02_Dispencers.fbDispencersDragLeftStation.tCycleTime;

P02_Dispencers.fbDispencer1.tCycleTime;
P02_Dispencers.fbDispencer2.tCycleTime;
P02_Dispencers.fbDispencer3.tCycleTime;
P02_Dispencers.fbDispencer4.tCycleTime;
P02_Dispencers.fbDispencerGatesStation.tCycleTime;
P02_Dispencers.fbDispencersCatch1Station.tCycleTime;
P02_Dispencers.fbDispencersCatch2Station.tCycleTime;
P02_Dispencers.fbDispencersCatch3Station.tCycleTime;
P02_Dispencers.fbDispencersCatch4Station.tCycleTime;


P05_Weight.fbWeight1.tCycleTime;
P05_Weight.fbWeight2.tCycleTime;
P05_Weight.fbWeight3.tCycleTime;
P05_Weight.fbWeight4.tCycleTime;


P09_CapPuttedCheck.fbCapPuttedCheck.tCycleTime;

P10_GripperScrewer.fb2GripperScrewer1.tCycleTime;
P10_GripperScrewer.fb2GripperScrewer2.tCycleTime;
P10_GripperScrewer.fbGripperScrewer1CatchStation.tCycleTime;
P10_GripperScrewer.fbGripperScrewer2CatchStation.tCycleTime;

P01_Gates.fbGateBeforeDispencers.tCycleTime;
P13_BottleTransfer.fbBottleTransfer.tCycleTime;




fbOEECycleTimes(
	bEnable:= TRUE, 
	bReset:= FALSE, 
	tStation1CT:= tMachineCycleTime, 
	bStation1En:= TRUE, 
	sStation1Name:= 'M', 
	tStation2CT:= P01_BottleFeeder.fbBottleFeeder.tCycleTime, 
	bStation2En:= P01_BottleFeeder.fbBottleFeeder.bEnable, 
	sStation2Name:= 'SORB', 
	tStation3CT:= P02_Dispencers.fbDispencersDragRightStation.tCycleTime , 
	bStation3En:= P02_Dispencers.fbDispencersDragRightStation.bEnable, 
	sStation3Name:= 'PFDP', 
	tStation4CT:= P02_Dispencers.fbDispencersDragLeftStation.tCycleTime, 
	bStation4En:= P02_Dispencers.fbDispencersDragLeftStation.bEnable, 
	sStation4Name:= 'PFDL', 
	tStation5CT:= P02_Dispencers.fbDispencer1.tCycleTime, 
	bStation5En:= P02_Dispencers.fbDispencer1.bEnable, 
	sStation5Name:= 'D1', 
	tStation6CT:= P02_Dispencers.fbDispencer2.tCycleTime, 
	bStation6En:= P02_Dispencers.fbDispencer2.bEnable,
	sStation6Name:= 'D2', 
	tStation7CT:= P02_Dispencers.fbDispencer3.tCycleTime, 
	bStation7En:= P02_Dispencers.fbDispencer3.bEnable, 
	sStation7Name:= 'D3', 
	tStation8CT:= P02_Dispencers.fbDispencer4.tCycleTime, 
	bStation8En:= P02_Dispencers.fbDispencer4.bEnable, 
	sStation8Name:= 'D4', 
	tStation9CT:= P02_Dispencers.fbDispencersCatch1Station.tCycleTime,
	bStation9En:= P02_Dispencers.fbDispencersCatch1Station.bEnable, 
	sStation9Name:= 'CHD1', 
	tStation10CT:= P02_Dispencers.fbDispencersCatch2Station.tCycleTime, 
	bStation10En:= P02_Dispencers.fbDispencersCatch2Station.bEnable, 
	sStation10Name:= 'CHD2', 
	tStation11CT:= P02_Dispencers.fbDispencersCatch3Station.tCycleTime, 
	bStation11En:= P02_Dispencers.fbDispencersCatch3Station.bEnable,
	sStation11Name:= 'CHD3', 
	tStation12CT:=  P02_Dispencers.fbDispencersCatch4Station.tCycleTime, 
	bStation12En:= P02_Dispencers.fbDispencersCatch4Station.bEnable, 
	sStation12Name:=  'CHD4', 
	tStation13CT:= P05_Weight.fbWeightStation.tCycleTime,
	bStation13En:= P05_Weight.fbWeightStation.bEnable, 
	sStation13Name:= 'PW',
	tStation14CT:= P05_Weight.fbWeightStation2Phase.tCycleTime,
	bStation14En:= P05_Weight.fbWeightStation2Phase.bEnable, 
	sStation14Name:= 'PW',	
	tStation15CT:= P05_Weight.fbWeight1.tCycleTime, 
	bStation15En:= P05_Weight.fbWeight1.bEnable, 
	sStation15Name:= 'W1', 
	tStation16CT:= P05_Weight.fbWeight2.tCycleTime, 
	bStation16En:= P05_Weight.fbWeight2.bEnable, 
	sStation16Name:= 'W2',  
	tStation17CT:= P05_Weight.fbWeight3.tCycleTime, 
	bStation17En:= P05_Weight.fbWeight3.bEnable, 
	sStation17Name:= 'W3',  
	tStation18CT:= P05_Weight.fbWeight4.tCycleTime, 
	bStation18En:= P05_Weight.fbWeight4.bEnable, 
	sStation18Name:= 'W4',  
	tStation19CT:= P05_Weight.fbWeight5.tCycleTime,  
	bStation19En:= P05_Weight.fbWeight5.bEnable,
	sStation19Name:= 'W5',
	tStation20CT:= P05_Weight.fbWeight6.tCycleTime,  
	bStation20En:= P05_Weight.fbWeight6.bEnable, 
	sStation20Name:= 'W6',  
	tStation21CT:= P10_GripperScrewer.fbGripperScrewersDragStation.tCycleTime, 
	bStation21En:= P10_GripperScrewer.fbGripperScrewersDragStation.bEnable,
	sStation21Name:= 'PFDZ',
	tStation22CT:= P10_GripperScrewer.fb2GripperScrewer1.tCycleTime, 
	bStation22En:= P10_GripperScrewer.fb2GripperScrewer1.bEnable1,
	sStation22Name:= 'ZS1',
	tStation23CT:= P10_GripperScrewer.fb2GripperScrewer2.tCycleTime, 
	bStation23En:= P10_GripperScrewer.fb2GripperScrewer2.bEnable2,
	sStation23Name:= 'ZS2',
	tStation24CT:= P10_GripperScrewer.fbGripperScrewersDragStation.tCycleTime, 
	bStation24En:= P10_GripperScrewer.fbGripperScrewersDragStation.bEnable,
	sStation24Name:= 'PFZ',
	tStation25CT:= P10_GripperScrewer.fbGripperScrewer1CatchStation.tCycleTime, 
	bStation25En:= P10_GripperScrewer.fbGripperScrewer1CatchStation.bEnable,
	sStation25Name:= 'CHZS1',
	tStation26CT:= P10_GripperScrewer.fbGripperScrewer2CatchStation.tCycleTime, 
	bStation26En:= P10_GripperScrewer.fbGripperScrewer2CatchStation.bEnable,
	sStation26Name:= 'CHZS2',
	tStation27CT:= P11_CapCorrectCheck.fbCapCorrectCheck.tCycleTime, 
	bStation27En:= P11_CapCorrectCheck.fbCapCorrectCheck.bEnable,
	sStation27Name:= 'SZA',
	tStation28CT:= P13_BottleTransfer.fbBottleTransfer.tCycleTime, 
	bStation28En:= P13_BottleTransfer.fbBottleTransfer.bEnable,
	sStation28Name:= 'R',  
	tStation29CT:= P01_Gates.fbGateBeforeDispencers.tCycleTime, 
	bStation29En:= P01_Gates.fbGateBeforeDispencers.bEnable, 
	sStation29Name:= 'SZD', 
	tStation20CT:= P01_Gates.fbGateRobot.tCycleTime, 
	bStation30En:= P01_Gates.fbGateRobot.bEnable, 
	sStation30Name:= 'SZR', 

	
	
	AsCycleTimes=> VIS.AsOEECycleTimes,
	
	
	
	);
END_ACTION

ACTION aMachinePartsChangeover:

VIS.bMachinePartsChangeOver	;						// Włączone przezbrajanie (ustawić z wizki)
VIS.iMachinePartsChangeOver	;						// Stan przezbrajania (0-ruch,1-pozycja gorna,-1-pozycja dolna) 
VIS.bBottleSorterDisable	;						// Wyłączenie sortera butelek
VIS.bCapSorterDisable		;						// Wyłączenie sortera nasadek


//Sygnał z wizki
VIS.bMachinePartsChangeover;
//Filtrowanie sygnału, przeciw lagom z wizualizacji lub ciągłym klikaniem
fbMachinePartsChangeover(bIn:=VIS.bMachinePartsChangeover,tFilterTimeOn:=T#3S,tFilterTimeOff:=T#3S,bOUT=>bChangeover);
//Przefiltrowany
bChangeover;

VIS.iMachinePartsChangeOver;
// Trzeba dodać, albo wyłączona stacja!
//Przezbrajanie - okienko 


IF bChangeover THEN
	VIS.bBottleSorterHold	:= TRUE;	
	VIS.bCapSorterHold		:= TRUE;	
	//VIS.bTank1SupplyPumpEnableShow:=FALSE;
	//VIS.bTank2SupplyPumpEnableShow:=FALSE;
ELSE
	//VIS.bBottleSorterHold	:= FALSE;	
	VIS.bCapSorterHold		:= FALSE;			
END_IF

IF 
 (P02_Dispencers.fbDispencersCatch1Station.eState = E_Station.ePreparingToDisable 			OR P02_Dispencers.fbDispencersCatch1Station.eState = E_Station.eHoming 				OR (NOT bDispencer1Enable AND NOT bDispencer3Enable)) 																			AND
 (P09_CapPuttedCheck.fbCapPuttedCheck.eState = E_Station.ePreparingToDisable				OR P09_CapPuttedCheck.fbCapPuttedCheck.eState = E_Station.eHoming				 	OR NOT bCapPuttedCheckEnable) 									AND
 (P10_GripperScrewer.fb2GripperScrewer1.eState = E_Station.ePreparingToDisable				OR P10_GripperScrewer.fb2GripperScrewer1.eState = E_Station.eHoming  				OR NOT bGripperScrewer1Enable) 									AND
 (P10_GripperScrewer.fb2GripperScrewer2.eState = E_Station.ePreparingToDisable				OR P10_GripperScrewer.fb2GripperScrewer2.eState = E_Station.eHoming  				OR NOT bGripperScrewer2Enable)									AND
 (P10_GripperScrewer.fbGripperScrewer1CatchStation.eState = E_Station.ePreparingToDisable 	OR P10_GripperScrewer.fbGripperScrewer1CatchStation.eState = E_Station.eHoming		OR NOT bGripperScrewer1Enable) 									AND
 (P10_GripperScrewer.fbGripperScrewer2CatchStation.eState = E_Station.ePreparingToDisable 	OR P10_GripperScrewer.fbGripperScrewer2CatchStation.eState = E_Station.eHoming 		OR NOT bGripperScrewer2Enable) 									AND
 (P11_CapCorrectCheck.fbCapCorrectCheck.eState = E_Station.ePreparingToDisable 				OR P11_CapCorrectCheck.fbCapCorrectCheck.eState = E_Station.eHoming					OR NOT bCapCorrectCheckEnable)
THEN
    VIS.iMachinePartsChangeOver := 0; //ruch
ELSIF
  (P02_Dispencers.fbDispencersCatch1Station.eState = E_Station.eDisabled			OR P02_Dispencers.fbDispencersCatch1Station.eState = E_Station.eManualMovement 			OR (NOT bDispencer1Enable AND NOT bDispencer3Enable) ) 											AND
 (P09_CapPuttedCheck.fbCapPuttedCheck.eState = E_Station.eDisabled				 	OR NOT bCapPuttedCheckEnable) 										AND
 (P10_GripperScrewer.fb2GripperScrewer1.eState = E_Station.eDisabled  				OR NOT bGripperScrewer1Enable)										AND
 (P10_GripperScrewer.fb2GripperScrewer2.eState = E_Station.eDisabled  				OR	NOT bGripperScrewer2Enable)										AND
 (P10_GripperScrewer.fbGripperScrewer1CatchStation.eState = E_Station.eDisabled 	OR NOT bGripperScrewer1Enable) 										AND
 (P10_GripperScrewer.fbGripperScrewer2CatchStation.eState = E_Station.eDisabled 	OR NOT bGripperScrewer2Enable) 										AND
 (P11_CapCorrectCheck.fbCapCorrectCheck.eState = E_Station.eDisabled 				OR NOT bCapCorrectCheckEnable)
THEN
    VIS.iMachinePartsChangeOver := 1; //1 pozycja gorna
ELSIF 
  (P02_Dispencers.fbDispencersCatch1Station.eState = E_Station.eReady 		OR P02_Dispencers.fbDispencersCatch1Station.eState = E_Station.eManualMovement 				OR (NOT bDispencer1Enable AND NOT bDispencer3Enable)) 												AND
 (P09_CapPuttedCheck.fbCapPuttedCheck.eState = E_Station.eReady				OR P09_CapPuttedCheck.fbCapPuttedCheck.eState = E_Station.eManualMovement			 		OR NOT bCapPuttedCheckEnable) 											AND
 (P10_GripperScrewer.fb2GripperScrewer1.eState = E_Station.eReady  			OR P10_GripperScrewer.fb2GripperScrewer1.eState = E_Station.eManualMovement					OR NOT bGripperScrewer1Enable)											AND
 (P10_GripperScrewer.fb2GripperScrewer2.eState = E_Station.eReady  			OR P10_GripperScrewer.fb2GripperScrewer2.eState = E_Station.eManualMovement					OR NOT bGripperScrewer2Enable) 											AND
 (P10_GripperScrewer.fbGripperScrewer1CatchStation.eState = E_Station.eReady OR P10_GripperScrewer.fbGripperScrewer1CatchStation.eState = E_Station.eManualMovement		OR NOT bGripperScrewer1Enable) 											AND
 (P10_GripperScrewer.fbGripperScrewer2CatchStation.eState = E_Station.eReady OR P10_GripperScrewer.fbGripperScrewer2CatchStation.eState = E_Station.eManualMovement		OR NOT bGripperScrewer2Enable) 											AND
 (P11_CapCorrectCheck.fbCapCorrectCheck.eState = E_Station.eReady 			OR	P11_CapCorrectCheck.fbCapCorrectCheck.eState = E_Station.eManualMovement 				OR NOT bCapCorrectCheckEnable)
THEN
    VIS.iMachinePartsChangeOver := -1; // -1pozycja dolna
END_IF 

//Kasowanie cyklu i liczników
rtChangeover(CLK:=bChangeover,Q=>);
IF rtChangeover.Q THEN
	//bCycleReseting := TRUE;	
	VIS.uiCounterAverageEfficiency:=0;
	VIS.udiCounterShiftBottles:=0;
	VIS.uiCounterInstantEfficiency:=0;
	VIS.uiCounterGoodBottles:=0;
	VIS.uiCounterBadBottles:=0;
END_IF
END_ACTION

ACTION aOEEPackMLSuspendedReason:
(*
Nazwa:			aOEEPackMLSuspendedReason
Wersja:			v0.1 			
Autor:			DP
Urzadzenia:		HMI, 
Konfiguracja:	
Info:
- Wyświetlanie na wykresie powodu zatrzymania lini, czyli w przyszłości przjeścia w stan PackML ->Suspended
Uwagi:

Zmiany:

*)
IF P00_PackML.tonCycleBadBottleConveyorFullSensor.Q THEN //odrzut
	VIS.iOEEPackMLSuspendedReason	:= 1;
ELSIF P16_LabelMachine.tonLabelMachineFullSensorInfo.Q THEN 
	//IF VIS.UPPackMLState=6 AND VIS.EPPackMLState=6 THEN		//etykieciarka
	VIS.iOEEPackMLSuspendedReason	:= 2;
ELSIF	vis.iMachineState = 2 OR vis.iMachineState = 8 OR vis.iMachineState = 9 OR vis.iMachineState = 15 THEN
	VIS.iOEEPackMLSuspendedReason	:= 3;
	//ELSIF VIS.UPPackMLState<>6 AND VIS.EPPackMLState=6 THEN //kartoniarka
	//VIS.iOEEPackMLSuspendedReason	:= 7;
	//ELSIF VIS.UPPackMLState=6 AND VIS.EPPackMLState<>6 THEN //paletyzer
	//VIS.iOEEPackMLSuspendedReason	:= 8;
	//END_IF
//ELSIF VIS.uliWarningOccure.33 THEN  //brak butelek
//	VIS.iOEEPackMLSuspendedReason	:= 3;	
//ELSIF VIS.uliWarningOccure.27 THEN	//brak nakrętek
//	VIS.iOEEPackMLSuspendedReason	:= 4;	
//(*ELSIF NOT P16_LabelMachine.tonLabelMachineFullSensorInfo.Q THEN		
//	IF VIS.UPPackMLState<>6 AND VIS.EPPackMLState=6 THEN			//kartoniarka
//	VIS.iOEEPackMLSuspendedReason	:= 7;
//	ELSIF VIS.UPPackMLState=6 AND VIS.EPPackMLState<>6 THEN			//paletyzer
//	VIS.iOEEPackMLSuspendedReason	:= 8;
//	END_IF*)
ELSE
	VIS.iOEEPackMLSuspendedReason	:= 0;		
END_IF
END_ACTION

ACTION aOEERaport:

//Data dla danych - według opisu
sOEEDateAndTime:= 
Concat(Concat(Concat(Concat(Concat(Concat(Concat(Concat(Concat(Concat(Concat(WORD_TO_STRING(wDay),'.'),WORD_TO_STRING(wMonth)),'.'),WORD_TO_STRING(wYear)),';'),WORD_TO_STRING(wHour)),':'),WORD_TO_STRING(wMinute)),';'),''),'');

//Generowanie raportu z wizki - podpiąć pod wybór receptury?
VIS.bOEEGenRaport;

//Zapisywanie daty wybrania receptury
//rtOEERaportChooseRecipe(CLK:=VIS.bChooseRecipe OR bOEETest1, Q=>);
rtOEERaportChooseRecipe(CLK:=VIS.bOEEGenRaport OR bOEETest1, Q=>);
tonbOEEGenRaport(IN:=VIS.bOEEGenRaport, PT:=T#500MS);
IF rtOEERaportChooseRecipe.Q THEN
	sOEEFileDateAndTime:= 
	Concat(Concat(Concat(Concat(Concat(Concat(Concat(Concat(Concat(Concat(Concat(WORD_TO_STRING(wYear),''),WORD_TO_STRING(wMonth)),''),WORD_TO_STRING(wDay)),''),WORD_TO_STRING(wHour)),''),WORD_TO_STRING(wMinute)),''),''),'');
	bOEETest1	:=	FALSE;
END_IF
IF tonbOEEGenRaport.Q THEN
	VIS.bOEEGenRaport	:= FALSE;
END_IF

//Zapisywanie danych co 1 min
rtOEERaportLogAddLine(CLK:=wMinute <> wOEERaportMinuteTemp, Q=>);	
IF rtOEERaportLogAddLine.Q THEN 
	wOEERaportMinuteTemp := wMinute;
END_IF

//Zapisywanie aktywnych bledow w stringu
IF rtOEERaportLogAddLine.Q THEN
	sOEEActiveErrorIDs := '';
	FOR i:=1 TO 10 DO
		IF VIS.fbAlarms.arrActiveEvents[i].stEventEntry.nEventId <> 0 THEN
			sOEEActiveErrorIDs:=Concat(sOEEActiveErrorIDs,Concat(UDINT_TO_STRING(VIS.fbAlarms.arrActiveEvents[i].stEventEntry.nEventId),';'));	
		END_IF
	END_FOR
	sOEEActiveErrorIDs:= Concat(sOEEActiveErrorIDs,stBottleSorterRead.eError.sStationName);
	sOEEActiveErrorIDs:= Concat(sOEEActiveErrorIDs,stCapSorterRead.eError.sStationName);	
END_IF			
		
//Raport nazwy,liczników itd
fbOEERaportLog(
	bExecute:= rtOEERaportLogAddLine.Q,
	AmsNetId:= , 
	sPath:='C:\Users\Administrator\Desktop\CSVFolder\', 
	sName:= Concat(sOEEFileDateAndTime,	Concat('-',Concat(sRecipeName,'.csv'))), 
	sLine:= 
	
Concat(
	'$R$N',
	Concat(
		sOEEDateAndTime,
		Concat(
				UINT_TO_STRING(VIS.iMachineState),
				Concat(
						';',
							Concat(
									sRecipeName,
									Concat(
											';',
											Concat(
													UDINT_TO_STRING(VIS.udiCounterGlobal),
														Concat(
																';',
																	Concat(
																		UDINT_TO_STRING(VIS.uiCounterBadBottles),
																		Concat(
																			';',
																			Concat(
																					//UDINT_TO_STRING(VIS.udiStationErrorCode),
																					sOEEActiveErrorIDs,
																					';'
																					)	
																				)	
																			)
																)
													)
											)
										)
						)
					)
				)
		)		
	,
	
	bBusy=>, 
	bError=>);

	IF rtOEERaportLogAddLine.Q THEN
		sOEEFRejectionLine := '';
		FOR i:= 0 TO 63 DO
			IF 	VIS.AStBadPackageReason[i].udiID <> 0 THEN
				
				sOEEFRejectionLine := 
					Concat(sOEEFRejectionLine,Concat(UDINT_TO_STRING(VIS.AStBadPackageReason[i].udiID), Concat(';',Concat(WSTRING_TO_STRING(VIS.AStBadPackageReason[i].wsDescription),';'))));
						
			END_IF
		END_FOR
	END_IF

//Raport odrzutów
fbOEERaportRejectionLog(
	bExecute:= rtOEERaportLogAddLine.Q,
	AmsNetId:= , 
	sPath:='C:\Users\Administrator\Desktop\CSVRejectionFolder\', 
	sName:= Concat(sOEEFileDateAndTime,	Concat('-',Concat(sRecipeName,'-Rejection.csv'))), 
	sLine:= Concat('$R$N',sOEEFRejectionLine),
	bBusy=>, 
	bError=>);
END_ACTION

ACTION aOEETime:

VIS.udiCounterShiftBottles;
VIS.udiCounterGlobal;            
VIS.udiCounterGlobalBadBottles;     

VIS.sOEEText1 := Concat(Concat('PRACA: ', UDINT_TO_STRING(udiCounterExecuteTimeTemp/60)),' min');
VIS.sOEEText2 := Concat(Concat('POSTÓJ: ', UDINT_TO_STRING(udiCounterReadyTimeTemp/60)),' min');
VIS.sOEEText3 := Concat(Concat('BŁĄD: ', UDINT_TO_STRING(udiCounterErrorTimeTemp/60)),' min');
tofIbBottleInFormCheckBottleSensor(IN:=MAIN.IbBottleInFormCheckBottleSensor,PT:=T#30S);

VIS.udiCounterExecuteTime	:=	UDINT_TO_UINT(udiCounterExecuteTimeTemp/60);
VIS.udiCounterReadyTime		:=	UDINT_TO_UINT(udiCounterReadyTimeTemp/60);
VIS.udiCounterErrorTime	  	:=	UDINT_TO_UINT(udiCounterErrorTimeTemp/60);
rtORRAdd1sec(CLK:=b2Hz,Q=>);

IF	
	//P00_PackML.fbPMLAuto.ePMLState = Tc3_PackML.E_PMLState.ePMLState_STARTING OR 
	//P00_PackML.fbPMLAuto.ePMLState = Tc3_PackML.E_PMLState.ePMLState_STOPPING OR 
	P00_PackML.fbPMLAuto.ePMLState = Tc3_PackML.E_PMLState.ePMLState_EXECUTE AND
	tofIbBottleInFormCheckBottleSensor.Q AND 
	NOT P16_LabelMachine.tonLabelMachineFullSensorInfo.Q AND
	NOT (P00_PackML.tonCycleBadBottleConveyorFullSensor.Q AND (P00_PackML.iRobotPickCase=110 OR P00_PackML.iRobotPickCase=210))
	THEN

	IF rtORRAdd1sec.Q THEN
		udiCounterExecuteTimeTemp	:=	udiCounterExecuteTimeTemp	+	1;
		
	END_IF
	
ELSIF
	P00_PackML.fbPMLAuto.ePMLState = Tc3_PackML.E_PMLState.ePMLState_STOPPED OR 
	P00_PackML.fbPMLAuto.ePMLState = Tc3_PackML.E_PMLState.ePMLState_ABORTED  
	THEN
	
	IF rtORRAdd1sec.Q THEN
		udiCounterErrorTimeTemp	:=	udiCounterErrorTimeTemp	+	1;
	END_IF	

ELSE
	IF rtORRAdd1sec.Q THEN
		udiCounterReadyTimeTemp	:=	udiCounterReadyTimeTemp	+	1;
	END_IF	
END_IF
END_ACTION

ACTION aRejectionReason:

//może uzależnić też od ilości opakowań do pobrania VIS.nBottleTransferPickOption			:=	1; // 1 butelka
//													VIS.nBottleTransferPlaceOption			:=	2; //Odrzucone butelki 

